LIN {X 0,Y 372.356,Z 524.558,A -85,B 0,C 180,E1 -12798.429,E2 -12798.429} C_VEL
LIN {X 0,Y 373.525,Z 512.398,A -85,B 0,C 180,E1 -12799.938,E2 -12799.938} C_VEL
LIN {X 0,Y 374.797,Z 499.165,A -85,B 0,C 180,E1 -12801.303,E2 -12801.303} C_VEL
LIN {X 0,Y 376.02,Z 484.644,A -85,B 0,C 180,E1 -12802.528,E2 -12802.528} C_VEL
LIN {X 0,Y 377.122,Z 470.65,A -85,B 0,C 180,E1 -12803.473,E2 -12803.473} C_VEL
LIN {X 0,Y 377.997,Z 455.018,A -85,B 0,C 180,E1 -12804.303,E2 -12804.303} C_VEL
LIN {X 0,Y 378.761,Z 440.368,A -85,B 0,C 180,E1 -12804.87,E2 -12804.87} C_VEL
LIN {X 0,Y 379.469,Z 417.557,A -85,B 0,C 180,E1 -12805.468,E2 -12805.468} C_VEL
LIN {X 0,Y 383.226,Z 310.701,A -85,B 0,C 180,E1 -12808.048,E2 -12808.048} C_VEL
LIN {X 0,Y 376.975,Z 295.774,A -85,B 0,C 180,E1 -12808.848,E2 -12808.848} C_VEL
LIN {X 0,Y 369.01,Z 277.788,A -85,B 0,C 180,E1 -12809.879,E2 -12809.879} C_VEL
LIN {X 0,Y 368.929,Z 277.156,A -85,B 0,C 180,E1 -12809.915,E2 -12809.915} C_VEL
LIN {X 0,Y 368.898,Z 277.158,A -85,B 0,C 180,E1 -12813.537,E2 -12813.537} C_VEL
LIN {X 0,Y 368.9,Z 277.154,A -85,B 0,C 180,E1 -12816.854,E2 -12816.854} C_VEL
LIN {X 0,Y 368.906,Z 277.155,A -85,B 0,C 180,E1 -12820.369,E2 -12820.369} C_VEL
LIN {X 0,Y 368.882,Z 277.161,A -85,B 0,C 180,E1 -12823.614,E2 -12823.614} C_VEL
LIN {X 0,Y 368.884,Z 277.157,A -85,B 0,C 180,E1 -12826.694,E2 -12826.694} C_VEL
LIN {X 0,Y 368.909,Z 277.158,A -85,B 0,C 180,E1 -12829.642,E2 -12829.642} C_VEL
LIN {X 0,Y 368.898,Z 277.156,A -85,B 0,C 180,E1 -12833.143,E2 -12833.143} C_VEL
LIN {X 0,Y 368.894,Z 277.156,A -85,B 0,C 180,E1 -12836.46,E2 -12836.46} C_VEL
LIN {X 0,Y 368.909,Z 277.154,A -85,B 0,C 180,E1 -12839.043,E2 -12839.043} C_VEL
LIN {X 0,Y 368.912,Z 277.158,A -85,B 0,C 180,E1 -12841.557,E2 -12841.557} C_VEL
LIN {X 0,Y 368.928,Z 277.153,A -85,B 0,C 180,E1 -12845.221,E2 -12845.221} C_VEL
LIN {X 0,Y 368.915,Z 277.153,A -85,B 0,C 180,E1 -12848.979,E2 -12848.979} C_VEL
LIN {X 0,Y 368.985,Z 277.145,A -85,B 0,C 180,E1 -12852.256,E2 -12852.256} C_VEL
LIN {X 0,Y 369.031,Z 277.139,A -85,B 0,C 180,E1 -12856.226,E2 -12856.226} C_VEL
LIN {X 0,Y 369.061,Z 277.136,A -85,B 0,C 180,E1 -12860.13,E2 -12860.13} C_VEL
LIN {X 0,Y 369.18,Z 277.12,A -85,B 0,C 180,E1 -12862.341,E2 -12862.341} C_VEL
LIN {X 0,Y 369.134,Z 277.125,A -85,B 0,C 180,E1 -12864.536,E2 -12864.536} C_VEL
LIN {X 0,Y 369.308,Z 277.108,A -85,B 0,C 180,E1 -12867.817,E2 -12867.817} C_VEL
LIN {X 0,Y 369.45,Z 277.088,A -85,B 0,C 180,E1 -12869.999,E2 -12869.999} C_VEL
LIN {X 0,Y 369.308,Z 277.105,A -85,B 0,C 180,E1 -12872.18,E2 -12872.18} C_VEL
LIN {X 0,Y 369.197,Z 277.117,A -85,B 0,C 180,E1 -12876.557,E2 -12876.557} C_VEL
LIN {X 0,Y 369.128,Z 277.126,A -85,B 0,C 180,E1 -12878.76,E2 -12878.76} C_VEL
LIN {X 0,Y 368.995,Z 277.144,A -85,B 0,C 180,E1 -12882.092,E2 -12882.092} C_VEL
LIN {X 0,Y 368.987,Z 277.15,A -85,B 0,C 180,E1 -12885.464,E2 -12885.464} C_VEL
LIN {X 0,Y 368.947,Z 277.15,A -85,B 0,C 180,E1 -12888.893,E2 -12888.893} C_VEL
LIN {X 0,Y 368.921,Z 277.155,A -85,B 0,C 180,E1 -12891.149,E2 -12891.149} C_VEL
LIN {X 0,Y 368.237,Z 277.247,A -85,B 0,C 180,E1 -12892.06,E2 -12892.06} C_VEL
LIN {X 0,Y 365.383,Z 277.603,A -85,B 0,C 180,E1 -12893.543,E2 -12893.543} C_VEL
LIN {X 0,Y 362.989,Z 277.896,A -85,B 0,C 180,E1 -12894.741,E2 -12894.741} C_VEL
LIN {X 0,Y 361.982,Z 278.02,A -85,B 0,C 180,E1 -12895.669,E2 -12895.669} C_VEL
LIN {X 0,Y 361.909,Z 278.025,A -85,B 0,C 180,E1 -12895.982,E2 -12895.982} C_VEL
LIN {X 0,Y 361.881,Z 278.032,A -85,B 0,C 180,E1 -12899.084,E2 -12899.084} C_VEL
LIN {X 0,Y 361.835,Z 278.037,A -85,B 0,C 180,E1 -12902.944,E2 -12902.944} C_VEL
LIN {X 0,Y 361.855,Z 278.035,A -85,B 0,C 180,E1 -12905.636,E2 -12905.636} C_VEL
LIN {X 0,Y 361.857,Z 278.035,A -85,B 0,C 180,E1 -12909.026,E2 -12909.026} C_VEL
LIN {X 0,Y 361.823,Z 278.038,A -85,B 0,C 180,E1 -12912.828,E2 -12912.828} C_VEL
LIN {X 0,Y 361.815,Z 278.038,A -85,B 0,C 180,E1 -12915.944,E2 -12915.944} C_VEL
LIN {X 0,Y 361.822,Z 278.043,A -85,B 0,C 180,E1 -12919.244,E2 -12919.244} C_VEL
LIN {X 0,Y 361.849,Z 278.035,A -85,B 0,C 180,E1 -12922.777,E2 -12922.777} C_VEL
LIN {X 0,Y 361.839,Z 278.036,A -85,B 0,C 180,E1 -12925.719,E2 -12925.719} C_VEL
LIN {X 0,Y 361.86,Z 278.033,A -85,B 0,C 180,E1 -12929.672,E2 -12929.672} C_VEL
LIN {X 0,Y 361.939,Z 278.025,A -85,B 0,C 180,E1 -12933.475,E2 -12933.475} C_VEL
LIN {X 0,Y 361.868,Z 278.037,A -85,B 0,C 180,E1 -12937.144,E2 -12937.144} C_VEL
LIN {X 0,Y 361.892,Z 278.03,A -85,B 0,C 180,E1 -12940.724,E2 -12940.724} C_VEL
LIN {X 0,Y 361.919,Z 278.03,A -85,B 0,C 180,E1 -12943.066,E2 -12943.066} C_VEL
LIN {X 0,Y 361.985,Z 278.017,A -85,B 0,C 180,E1 -12946.528,E2 -12946.528} C_VEL
LIN {X 0,Y 362.017,Z 278.012,A -85,B 0,C 180,E1 -12949.939,E2 -12949.939} C_VEL
LIN {X 0,Y 362.147,Z 277.999,A -85,B 0,C 180,E1 -12953.314,E2 -12953.314} C_VEL
LIN {X 0,Y 362.269,Z 277.981,A -85,B 0,C 180,E1 -12957.777,E2 -12957.777} C_VEL
LIN {X 0,Y 362.415,Z 277.962,A -85,B 0,C 180,E1 -12960.001,E2 -12960.001} C_VEL
LIN {X 0,Y 362.267,Z 277.981,A -85,B 0,C 180,E1 -12962.224,E2 -12962.224} C_VEL
LIN {X 0,Y 362.158,Z 277.998,A -85,B 0,C 180,E1 -12966.687,E2 -12966.687} C_VEL
LIN {X 0,Y 362.062,Z 278.013,A -85,B 0,C 180,E1 -12968.934,E2 -12968.934} C_VEL
LIN {X 0,Y 361.948,Z 278.021,A -85,B 0,C 180,E1 -12972.333,E2 -12972.333} C_VEL
LIN {X 0,Y 361.951,Z 278.023,A -85,B 0,C 180,E1 -12974.622,E2 -12974.622} C_VEL
LIN {X 0,Y 361.945,Z 278.021,A -85,B 0,C 180,E1 -12978.101,E2 -12978.101} C_VEL
LIN {X 0,Y 361.851,Z 278.033,A -85,B 0,C 180,E1 -12981.656,E2 -12981.656} C_VEL
LIN {X 0,Y 361.917,Z 278.027,A -85,B 0,C 180,E1 -12985.292,E2 -12985.292} C_VEL
LIN {X 0,Y 361.904,Z 278.026,A -85,B 0,C 180,E1 -12987.78,E2 -12987.78} C_VEL
LIN {X 0,Y 361.837,Z 278.036,A -85,B 0,C 180,E1 -12991.287,E2 -12991.287} C_VEL
LIN {X 0,Y 361.846,Z 278.035,A -85,B 0,C 180,E1 -12994.282,E2 -12994.282} C_VEL
LIN {X 0,Y 361.855,Z 278.034,A -85,B 0,C 180,E1 -12997.224,E2 -12997.224} C_VEL
LIN {X 0,Y 361.828,Z 278.042,A -85,B 0,C 180,E1 -13000.757,E2 -13000.757} C_VEL
LIN {X 0,Y 361.838,Z 278.037,A -85,B 0,C 180,E1 -13004.366,E2 -13004.366} C_VEL
LIN {X 0,Y 361.83,Z 278.035,A -85,B 0,C 180,E1 -13007.57,E2 -13007.57} C_VEL
LIN {X 0,Y 361.864,Z 278.036,A -85,B 0,C 180,E1 -13010.975,E2 -13010.975} C_VEL
LIN {X 0,Y 361.867,Z 278.117,A -85,B 0,C 180,E1 -13012.777,E2 -13012.777} C_VEL
LIN {X 0,Y 365.951,Z 294.107,A -85,B 0,C 180,E1 -13016.158,E2 -13016.158} C_VEL
LIN {X 0,Y 369.838,Z 310.572,A -85,B 0,C 180,E1 -13019.45,E2 -13019.45} C_VEL
LIN {X 0,Y 369.826,Z 313.182,A -85,B 0,C 180,E1 -13019.922,E2 -13019.922} C_VEL
LIN {X 0,Y 376.375,Z 356.911,A -85,B 0,C 180,E1 -13021.56,E2 -13021.56} C_VEL
LIN {X 0,Y 371.811,Z 479.859,A -85,B 0,C 180,E1 -13024.645,E2 -13024.645} C_VEL
LIN {X 0,Y 370.896,Z 495.184,A -85,B 0,C 180,E1 -13025.215,E2 -13025.215} C_VEL
LIN {X 0,Y 369.768,Z 509.984,A -85,B 0,C 180,E1 -13025.971,E2 -13025.971} C_VEL
LIN {X 0,Y 368.493,Z 525.199,A -85,B 0,C 180,E1 -13026.986,E2 -13026.986} C_VEL
LIN {X 0,Y 367.201,Z 538.472,A -85,B 0,C 180,E1 -13028.088,E2 -13028.088} C_VEL
LIN {X 0,Y 365.807,Z 552.139,A -85,B 0,C 180,E1 -13029.476,E2 -13029.476} C_VEL
LIN {X 0,Y 364.498,Z 564.433,A -85,B 0,C 180,E1 -13030.983,E2 -13030.983} C_VEL
LIN {X 0,Y 363.421,Z 575.247,A -85,B 0,C 180,E1 -13032.559,E2 -13032.559} C_VEL
LIN {X 0,Y 362.424,Z 585.017,A -85,B 0,C 180,E1 -13034.249,E2 -13034.249} C_VEL
LIN {X 0,Y 361.728,Z 593.578,A -85,B 0,C 180,E1 -13036.004,E2 -13036.004} C_VEL
LIN {X 0,Y 361.109,Z 601.45,A -85,B 0,C 180,E1 -13037.925,E2 -13037.925} C_VEL
LIN {X 0,Y 360.725,Z 608.122,A -85,B 0,C 180,E1 -13039.903,E2 -13039.903} C_VEL
LIN {X 0,Y 360.555,Z 614.167,A -85,B 0,C 180,E1 -13042.159,E2 -13042.159} C_VEL
LIN {X 0,Y 360.492,Z 618.678,A -85,B 0,C 180,E1 -13044.408,E2 -13044.408} C_VEL
LIN {X 0,Y 360.435,Z 621.759,A -85,B 0,C 180,E1 -13046.648,E2 -13046.648} C_VEL
LIN {X 0,Y 360.564,Z 622.799,A -85,B 0,C 180,E1 -13047.767,E2 -13047.767} C_VEL
LIN {X 0,Y 360.519,Z 623.861,A -85,B 0,C 180,E1 -13050.002,E2 -13050.002} C_VEL
LIN {X 0,Y 360.491,Z 623.607,A -85,B 0,C 180,E1 -13052.236,E2 -13052.236} C_VEL
LIN {X 0,Y 360.403,Z 622.015,A -85,B 0,C 180,E1 -13054.475,E2 -13054.475} C_VEL
LIN {X 0,Y 360.395,Z 619.123,A -85,B 0,C 180,E1 -13056.721,E2 -13056.721} C_VEL
LIN {X 0,Y 360.566,Z 614.896,A -85,B 0,C 180,E1 -13058.972,E2 -13058.972} C_VEL
LIN {X 0,Y 361,Z 609.253,A -85,B 0,C 180,E1 -13061.228,E2 -13061.228} C_VEL
LIN {X 0,Y 361.677,Z 602.075,A -85,B 0,C 180,E1 -13063.486,E2 -13063.486} C_VEL
LIN {X 0,Y 362.806,Z 593.186,A -85,B 0,C 180,E1 -13065.737,E2 -13065.737} C_VEL
LIN {X 0,Y 364.158,Z 583.775,A -85,B 0,C 180,E1 -13067.697,E2 -13067.697} C_VEL
LIN {X 0,Y 365.645,Z 573.556,A -85,B 0,C 180,E1 -13069.491,E2 -13069.491} C_VEL
LIN {X 0,Y 367.627,Z 561.225,A -85,B 0,C 180,E1 -13071.3,E2 -13071.3} C_VEL
LIN {X 0,Y 369.765,Z 547.82,A -85,B 0,C 180,E1 -13072.933,E2 -13072.933} C_VEL
LIN {X 0,Y 372.055,Z 533.098,A -85,B 0,C 180,E1 -13074.408,E2 -13074.408} C_VEL
LIN {X 0,Y 374.237,Z 518.489,A -85,B 0,C 180,E1 -13075.591,E2 -13075.591} C_VEL
LIN {X 0,Y 376.417,Z 502.554,A -85,B 0,C 180,E1 -13076.623,E2 -13076.623} C_VEL
LIN {X 0,Y 378.583,Z 485.245,A -85,B 0,C 180,E1 -13077.466,E2 -13077.466} C_VEL
LIN {X 0,Y 380.092,Z 468.909,A -85,B 0,C 180,E1 -13078.058,E2 -13078.058} C_VEL
LIN {X 0,Y 385.883,Z 394.775,A -85,B 0,C 180,E1 -13080.322,E2 -13080.322} C_VEL
LIN {X 0,Y 389.106,Z 358.696,A -85,B 0,C 180,E1 -13081.484,E2 -13081.484} C_VEL
LIN {X 0,Y 388.296,Z 346.311,A -85,B 0,C 180,E1 -13082.234,E2 -13082.234} C_VEL
LIN {X 0,Y 386.535,Z 330.75,A -85,B 0,C 180,E1 -13083.397,E2 -13083.397} C_VEL
LIN {X 0,Y 383.665,Z 323.796,A -85,B 0,C 180,E1 -13084.421,E2 -13084.421} C_VEL
LIN {X 0,Y 381.231,Z 318.55,A -85,B 0,C 180,E1 -13085.337,E2 -13085.337} C_VEL
LIN {X 0,Y 378.301,Z 312.803,A -85,B 0,C 180,E1 -13086.548,E2 -13086.548} C_VEL
LIN {X 0,Y 374.397,Z 305.694,A -85,B 0,C 180,E1 -13088.473,E2 -13088.473} C_VEL
LIN {X 0,Y 370.905,Z 299.971,A -85,B 0,C 180,E1 -13090.782,E2 -13090.782} C_VEL
LIN {X 0,Y 369.189,Z 296.566,A -85,B 0,C 180,E1 -13092.669,E2 -13092.669} C_VEL
LIN {X 0,Y 368.787,Z 295.464,A -85,B 0,C 180,E1 -13093.6,E2 -13093.6} C_VEL
LIN {X 0,Y 368.258,Z 294.192,A -85,B 0,C 180,E1 -13095.439,E2 -13095.439} C_VEL
LIN {X 0,Y 368.708,Z 294.364,A -85,B 0,C 180,E1 -13097.364,E2 -13097.364} C_VEL
LIN {X 0,Y 370.91,Z 296.011,A -85,B 0,C 180,E1 -13099.891,E2 -13099.891} C_VEL
LIN {X 0,Y 372.199,Z 297.038,A -85,B 0,C 180,E1 -13100.825,E2 -13100.825} C_VEL
LIN {X 0,Y 375.738,Z 300.987,A -85,B 0,C 180,E1 -13102.863,E2 -13102.863} C_VEL
LIN {X 0,Y 379.159,Z 305.289,A -85,B 0,C 180,E1 -13104.391,E2 -13104.391} C_VEL
LIN {X 0,Y 382.506,Z 310.037,A -85,B 0,C 180,E1 -13105.673,E2 -13105.673} C_VEL
LIN {X 0,Y 386.077,Z 315.376,A -85,B 0,C 180,E1 -13106.865,E2 -13106.865} C_VEL
LIN {X 0,Y 390.641,Z 323.626,A -85,B 0,C 180,E1 -13108.26,E2 -13108.26} C_VEL
LIN {X 0,Y 391.487,Z 325.432,A -85,B 0,C 180,E1 -13108.513,E2 -13108.513} C_VEL
LIN {X 0,Y 383.852,Z 405.157,A -85,B 0,C 180,E1 -13111.049,E2 -13111.049} C_VEL
LIN {X 0,Y 380.62,Z 447.423,A -85,B 0,C 180,E1 -13112.387,E2 -13112.387} C_VEL
LIN {X 0,Y 379.204,Z 462.75,A -85,B 0,C 180,E1 -13113.077,E2 -13113.077} C_VEL
LIN {X 0,Y 377.435,Z 478.879,A -85,B 0,C 180,E1 -13114.05,E2 -13114.05} C_VEL
LIN {X 0,Y 375.724,Z 492.725,A -85,B 0,C 180,E1 -13115.11,E2 -13115.11} C_VEL
LIN {X 0,Y 373.879,Z 505.632,A -85,B 0,C 180,E1 -13116.309,E2 -13116.309} C_VEL
LIN {X 0,Y 371.825,Z 518.795,A -85,B 0,C 180,E1 -13117.788,E2 -13117.788} C_VEL
LIN {X 0,Y 370.029,Z 528.933,A -85,B 0,C 180,E1 -13119.137,E2 -13119.137} C_VEL
LIN {X 0,Y 368.265,Z 539.317,A -85,B 0,C 180,E1 -13120.779,E2 -13120.779} C_VEL
LIN {X 0,Y 366.473,Z 549.487,A -85,B 0,C 180,E1 -13122.707,E2 -13122.707} C_VEL
LIN {X 0,Y 364.854,Z 557.896,A -85,B 0,C 180,E1 -13124.624,E2 -13124.624} C_VEL
LIN {X 0,Y 363.668,Z 564.97,A -85,B 0,C 180,E1 -13126.59,E2 -13126.59} C_VEL
LIN {X 0,Y 362.517,Z 571.438,A -85,B 0,C 180,E1 -13128.821,E2 -13128.821} C_VEL
LIN {X 0,Y 361.765,Z 576.407,A -85,B 0,C 180,E1 -13131.058,E2 -13131.058} C_VEL
LIN {X 0,Y 361.195,Z 580.029,A -85,B 0,C 180,E1 -13133.295,E2 -13133.295} C_VEL
LIN {X 0,Y 360.877,Z 582.365,A -85,B 0,C 180,E1 -13135.531,E2 -13135.531} C_VEL
LIN {X 0,Y 360.694,Z 583.454,A -85,B 0,C 180,E1 -13137.766,E2 -13137.766} C_VEL
LIN {X 0,Y 360.524,Z 583.282,A -85,B 0,C 180,E1 -13139.999,E2 -13139.999} C_VEL
LIN {X 0,Y 360.61,Z 581.862,A -85,B 0,C 180,E1 -13142.233,E2 -13142.233} C_VEL
LIN {X 0,Y 360.609,Z 579.19,A -85,B 0,C 180,E1 -13144.47,E2 -13144.47} C_VEL
LIN {X 0,Y 360.827,Z 574.99,A -85,B 0,C 180,E1 -13146.806,E2 -13146.806} C_VEL
LIN {X 0,Y 361.116,Z 569.776,A -85,B 0,C 180,E1 -13148.956,E2 -13148.956} C_VEL
LIN {X 0,Y 361.608,Z 562.801,A -85,B 0,C 180,E1 -13151.206,E2 -13151.206} C_VEL
LIN {X 0,Y 362.378,Z 555.243,A -85,B 0,C 180,E1 -13153.171,E2 -13153.171} C_VEL
LIN {X 0,Y 363.207,Z 546.104,A -85,B 0,C 180,E1 -13155.142,E2 -13155.142} C_VEL
LIN {X 0,Y 364.364,Z 535.081,A -85,B 0,C 180,E1 -13157.105,E2 -13157.105} C_VEL
LIN {X 0,Y 365.534,Z 523.732,A -85,B 0,C 180,E1 -13158.786,E2 -13158.786} C_VEL
LIN {X 0,Y 366.761,Z 511.326,A -85,B 0,C 180,E1 -13160.322,E2 -13160.322} C_VEL
LIN {X 0,Y 368.079,Z 497.791,A -85,B 0,C 180,E1 -13161.711,E2 -13161.711} C_VEL
LIN {X 0,Y 369.19,Z 484.653,A -85,B 0,C 180,E1 -13162.82,E2 -13162.82} C_VEL
LIN {X 0,Y 370.313,Z 470.577,A -85,B 0,C 180,E1 -13163.783,E2 -13163.783} C_VEL
LIN {X 0,Y 371.208,Z 455.124,A -85,B 0,C 180,E1 -13164.614,E2 -13164.614} C_VEL
LIN {X 0,Y 372.028,Z 439.672,A -85,B 0,C 180,E1 -13165.216,E2 -13165.216} C_VEL
LIN {X 0,Y 372.982,Z 410.158,A -85,B 0,C 180,E1 -13165.981,E2 -13165.981} C_VEL
LIN {X 0,Y 376.663,Z 312.659,A -85,B 0,C 180,E1 -13168.402,E2 -13168.402} C_VEL
LIN {X 0,Y 371.332,Z 299.862,A -85,B 0,C 180,E1 -13169.098,E2 -13169.098} C_VEL
LIN {X 0,Y 361.953,Z 278.543,A -85,B 0,C 180,E1 -13170.344,E2 -13170.344} C_VEL
LIN {X 0,Y 361.888,Z 278.033,A -85,B 0,C 180,E1 -13170.402,E2 -13170.402} C_VEL
LIN {X 0,Y 361.855,Z 278.035,A -85,B 0,C 180,E1 -13174.279,E2 -13174.279} C_VEL
LIN {X 0,Y 361.861,Z 278.032,A -85,B 0,C 180,E1 -13177.221,E2 -13177.221} C_VEL
LIN {X 0,Y 361.829,Z 278.035,A -85,B 0,C 180,E1 -13180.753,E2 -13180.753} C_VEL
LIN {X 0,Y 361.816,Z 278.038,A -85,B 0,C 180,E1 -13184.367,E2 -13184.367} C_VEL
LIN {X 0,Y 361.835,Z 278.038,A -85,B 0,C 180,E1 -13187.566,E2 -13187.566} C_VEL
LIN {X 0,Y 361.866,Z 278.031,A -85,B 0,C 180,E1 -13190.972,E2 -13190.972} C_VEL
LIN {X 0,Y 361.871,Z 278.03,A -85,B 0,C 180,E1 -13194.654,E2 -13194.654} C_VEL
LIN {X 0,Y 361.834,Z 278.036,A -85,B 0,C 180,E1 -13198.369,E2 -13198.369} C_VEL
LIN {X 0,Y 361.862,Z 278.032,A -85,B 0,C 180,E1 -13200.95,E2 -13200.95} C_VEL
LIN {X 0,Y 361.886,Z 278.028,A -85,B 0,C 180,E1 -13204.705,E2 -13204.705} C_VEL
LIN {X 0,Y 361.856,Z 278.033,A -85,B 0,C 180,E1 -13208.343,E2 -13208.343} C_VEL
LIN {X 0,Y 361.915,Z 278.027,A -85,B 0,C 180,E1 -13212.083,E2 -13212.083} C_VEL
LIN {X 0,Y 361.956,Z 278.023,A -85,B 0,C 180,E1 -13215.378,E2 -13215.378} C_VEL
LIN {X 0,Y 361.965,Z 278.019,A -85,B 0,C 180,E1 -13218.803,E2 -13218.803} C_VEL
LIN {X 0,Y 362.143,Z 277.997,A -85,B 0,C 180,E1 -13222.191,E2 -13222.191} C_VEL
LIN {X 0,Y 362.108,Z 278.001,A -85,B 0,C 180,E1 -13224.43,E2 -13224.43} C_VEL
LIN {X 0,Y 362.272,Z 277.984,A -85,B 0,C 180,E1 -13227.775,E2 -13227.775} C_VEL
LIN {X 0,Y 362.419,Z 277.964,A -85,B 0,C 180,E1 -13229.998,E2 -13229.998} C_VEL
LIN {X 0,Y 362.272,Z 277.981,A -85,B 0,C 180,E1 -13232.222,E2 -13232.222} C_VEL
LIN {X 0,Y 362.161,Z 277.994,A -85,B 0,C 180,E1 -13236.685,E2 -13236.685} C_VEL
LIN {X 0,Y 362.064,Z 278.007,A -85,B 0,C 180,E1 -13238.932,E2 -13238.932} C_VEL
LIN {X 0,Y 361.95,Z 278.02,A -85,B 0,C 180,E1 -13242.331,E2 -13242.331} C_VEL
LIN {X 0,Y 361.951,Z 278.02,A -85,B 0,C 180,E1 -13244.619,E2 -13244.619} C_VEL
LIN {X 0,Y 361.945,Z 278.022,A -85,B 0,C 180,E1 -13248.098,E2 -13248.098} C_VEL
LIN {X 0,Y 361.882,Z 278.033,A -85,B 0,C 180,E1 -13251.652,E2 -13251.652} C_VEL
LIN {X 0,Y 361.916,Z 278.03,A -85,B 0,C 180,E1 -13255.289,E2 -13255.289} C_VEL
LIN {X 0,Y 361.909,Z 278.025,A -85,B 0,C 180,E1 -13255.982,E2 -13255.982} C_VEL
LIN {X 0,Y 361.251,Z 278.111,A -85,B 0,C 180,E1 -13256.911,E2 -13256.911} C_VEL
LIN {X 0,Y 358.342,Z 278.47,A -85,B 0,C 180,E1 -13258.42,E2 -13258.42} C_VEL
LIN {X 0,Y 355.883,Z 278.78,A -85,B 0,C 180,E1 -13259.642,E2 -13259.642} C_VEL
LIN {X 0,Y 354.851,Z 278.905,A -85,B 0,C 180,E1 -13260.588,E2 -13260.588} C_VEL
LIN {X 0,Y 354.782,Z 278.915,A -85,B 0,C 180,E1 -13260.908,E2 -13260.908} C_VEL
LIN {X 0,Y 354.793,Z 278.915,A -85,B 0,C 180,E1 -13263.701,E2 -13263.701} C_VEL
LIN {X 0,Y 354.787,Z 278.913,A -85,B 0,C 180,E1 -13266.458,E2 -13266.458} C_VEL
LIN {X 0,Y 354.81,Z 278.915,A -85,B 0,C 180,E1 -13269.423,E2 -13269.423} C_VEL
LIN {X 0,Y 354.775,Z 278.916,A -85,B 0,C 180,E1 -13272.867,E2 -13272.867} C_VEL
LIN {X 0,Y 354.762,Z 278.916,A -85,B 0,C 180,E1 -13276.105,E2 -13276.105} C_VEL
LIN {X 0,Y 354.774,Z 278.92,A -85,B 0,C 180,E1 -13279.179,E2 -13279.179} C_VEL
LIN {X 0,Y 354.793,Z 278.912,A -85,B 0,C 180,E1 -13282.402,E2 -13282.402} C_VEL
LIN {X 0,Y 354.797,Z 278.915,A -85,B 0,C 180,E1 -13284.941,E2 -13284.941} C_VEL
LIN {X 0,Y 354.778,Z 278.914,A -85,B 0,C 180,E1 -13288.405,E2 -13288.405} C_VEL
LIN {X 0,Y 354.835,Z 278.909,A -85,B 0,C 180,E1 -13291.619,E2 -13291.619} C_VEL
LIN {X 0,Y 354.884,Z 278.9,A -85,B 0,C 180,E1 -13294.173,E2 -13294.173} C_VEL
LIN {X 0,Y 354.802,Z 278.911,A -85,B 0,C 180,E1 -13297.893,E2 -13297.893} C_VEL
LIN {X 0,Y 354.908,Z 278.898,A -85,B 0,C 180,E1 -13301.892,E2 -13301.892} C_VEL
LIN {X 0,Y 354.929,Z 278.895,A -85,B 0,C 180,E1 -13305.982,E2 -13305.982} C_VEL
LIN {X 0,Y 354.964,Z 278.891,A -85,B 0,C 180,E1 -13309.737,E2 -13309.737} C_VEL
LIN {X 0,Y 355.111,Z 278.877,A -85,B 0,C 180,E1 -13313.181,E2 -13313.181} C_VEL
LIN {X 0,Y 355.232,Z 278.858,A -85,B 0,C 180,E1 -13317.733,E2 -13317.733} C_VEL
LIN {X 0,Y 355.385,Z 278.838,A -85,B 0,C 180,E1 -13320.001,E2 -13320.001} C_VEL
LIN {X 0,Y 355.23,Z 278.858,A -85,B 0,C 180,E1 -13322.269,E2 -13322.269} C_VEL
LIN {X 0,Y 355.124,Z 278.875,A -85,B 0,C 180,E1 -13326.82,E2 -13326.82} C_VEL
LIN {X 0,Y 355.004,Z 278.89,A -85,B 0,C 180,E1 -13329.113,E2 -13329.113} C_VEL
LIN {X 0,Y 354.91,Z 278.9,A -85,B 0,C 180,E1 -13332.582,E2 -13332.582} C_VEL
LIN {X 0,Y 354.878,Z 278.901,A -85,B 0,C 180,E1 -13336.097,E2 -13336.097} C_VEL
LIN {X 0,Y 354.891,Z 278.902,A -85,B 0,C 180,E1 -13338.473,E2 -13338.473} C_VEL
LIN {X 0,Y 354.807,Z 278.91,A -85,B 0,C 180,E1 -13342.109,E2 -13342.109} C_VEL
LIN {X 0,Y 354.889,Z 278.9,A -85,B 0,C 180,E1 -13345.829,E2 -13345.829} C_VEL
LIN {X 0,Y 354.845,Z 278.906,A -85,B 0,C 180,E1 -13349.68,E2 -13349.68} C_VEL
LIN {X 0,Y 354.798,Z 278.911,A -85,B 0,C 180,E1 -13353.704,E2 -13353.704} C_VEL
LIN {X 0,Y 354.789,Z 278.915,A -85,B 0,C 180,E1 -13356.461,E2 -13356.461} C_VEL
LIN {X 0,Y 354.817,Z 278.91,A -85,B 0,C 180,E1 -13359.425,E2 -13359.425} C_VEL
LIN {X 0,Y 354.781,Z 278.919,A -85,B 0,C 180,E1 -13362.869,E2 -13362.869} C_VEL
LIN {X 0,Y 354.762,Z 278.917,A -85,B 0,C 180,E1 -13366.106,E2 -13366.106} C_VEL
LIN {X 0,Y 354.782,Z 278.918,A -85,B 0,C 180,E1 -13369.181,E2 -13369.181} C_VEL
LIN {X 0,Y 354.847,Z 278.966,A -85,B 0,C 180,E1 -13372.361,E2 -13372.361} C_VEL
LIN {X 0,Y 359.247,Z 296.405,A -85,B 0,C 180,E1 -13376.116,E2 -13376.116} C_VEL
LIN {X 0,Y 362.932,Z 311.997,A -85,B 0,C 180,E1 -13379.288,E2 -13379.288} C_VEL
LIN {X 0,Y 363.077,Z 313.226,A -85,B 0,C 180,E1 -13379.472,E2 -13379.472} C_VEL
LIN {X 0,Y 369.741,Z 357.719,A -85,B 0,C 180,E1 -13381.181,E2 -13381.181} C_VEL
LIN {X 0,Y 365.017,Z 479.813,A -85,B 0,C 180,E1 -13384.33,E2 -13384.33} C_VEL
LIN {X 0,Y 363.984,Z 496.194,A -85,B 0,C 180,E1 -13384.968,E2 -13384.968} C_VEL
LIN {X 0,Y 362.839,Z 511.005,A -85,B 0,C 180,E1 -13385.761,E2 -13385.761} C_VEL
LIN {X 0,Y 361.493,Z 526.191,A -85,B 0,C 180,E1 -13386.818,E2 -13386.818} C_VEL
LIN {X 0,Y 360.19,Z 539.216,A -85,B 0,C 180,E1 -13387.94,E2 -13387.94} C_VEL
LIN {X 0,Y 358.772,Z 552.689,A -85,B 0,C 180,E1 -13389.355,E2 -13389.355} C_VEL
LIN {X 0,Y 357.382,Z 565.219,A -85,B 0,C 180,E1 -13390.945,E2 -13390.945} C_VEL
LIN {X 0,Y 356.327,Z 575.531,A -85,B 0,C 180,E1 -13392.497,E2 -13392.497} C_VEL
LIN {X 0,Y 355.332,Z 585.239,A -85,B 0,C 180,E1 -13394.221,E2 -13394.221} C_VEL
LIN {X 0,Y 354.5,Z 594.861,A -85,B 0,C 180,E1 -13396.273,E2 -13396.273} C_VEL
LIN {X 0,Y 353.985,Z 602.563,A -85,B 0,C 180,E1 -13398.26,E2 -13398.26} C_VEL
LIN {X 0,Y 353.594,Z 608.931,A -85,B 0,C 180,E1 -13400.275,E2 -13400.275} C_VEL
LIN {X 0,Y 353.48,Z 613.391,A -85,B 0,C 180,E1 -13402.001,E2 -13402.001} C_VEL
LIN {X 0,Y 353.43,Z 618.004,A -85,B 0,C 180,E1 -13404.296,E2 -13404.296} C_VEL
LIN {X 0,Y 353.348,Z 621.175,A -85,B 0,C 180,E1 -13406.581,E2 -13406.581} C_VEL
LIN {X 0,Y 353.482,Z 622.259,A -85,B 0,C 180,E1 -13407.723,E2 -13407.723} C_VEL
LIN {X 0,Y 353.454,Z 623.4,A -85,B 0,C 180,E1 -13410.002,E2 -13410.002} C_VEL
LIN {X 0,Y 353.467,Z 623.464,A -85,B 0,C 180,E1 -13411.141,E2 -13411.141} C_VEL
LIN {X 0,Y 353.305,Z 622.586,A -85,B 0,C 180,E1 -13413.423,E2 -13413.423} C_VEL
LIN {X 0,Y 353.312,Z 620.419,A -85,B 0,C 180,E1 -13415.71,E2 -13415.71} C_VEL
LIN {X 0,Y 353.396,Z 616.945,A -85,B 0,C 180,E1 -13418.004,E2 -13418.004} C_VEL
LIN {X 0,Y 353.647,Z 612.107,A -85,B 0,C 180,E1 -13420.305,E2 -13420.305} C_VEL
LIN {X 0,Y 354.276,Z 605.801,A -85,B 0,C 180,E1 -13422.606,E2 -13422.606} C_VEL
LIN {X 0,Y 355.257,Z 597.902,A -85,B 0,C 180,E1 -13424.904,E2 -13424.904} C_VEL
LIN {X 0,Y 356.476,Z 589.531,A -85,B 0,C 180,E1 -13426.907,E2 -13426.907} C_VEL
LIN {X 0,Y 358.053,Z 579.559,A -85,B 0,C 180,E1 -13428.898,E2 -13428.898} C_VEL
LIN {X 0,Y 360.045,Z 567.668,A -85,B 0,C 180,E1 -13430.871,E2 -13430.871} C_VEL
LIN {X 0,Y 362.343,Z 554.497,A -85,B 0,C 180,E1 -13432.676,E2 -13432.676} C_VEL
LIN {X 0,Y 364.583,Z 541.247,A -85,B 0,C 180,E1 -13434.183,E2 -13434.183} C_VEL
LIN {X 0,Y 366.859,Z 527.358,A -85,B 0,C 180,E1 -13435.493,E2 -13435.493} C_VEL
LIN {X 0,Y 369.401,Z 511.331,A -85,B 0,C 180,E1 -13436.711,E2 -13436.711} C_VEL
LIN {X 0,Y 371.72,Z 495.021,A -85,B 0,C 180,E1 -13437.672,E2 -13437.672} C_VEL
LIN {X 0,Y 373.743,Z 478.107,A -85,B 0,C 180,E1 -13438.425,E2 -13438.425} C_VEL
LIN {X 0,Y 376.103,Z 449.941,A -85,B 0,C 180,E1 -13439.338,E2 -13439.338} C_VEL
LIN {X 0,Y 382.639,Z 377.508,A -85,B 0,C 180,E1 -13441.652,E2 -13441.652} C_VEL
LIN {X 0,Y 384.308,Z 359.927,A -85,B 0,C 180,E1 -13442.25,E2 -13442.25} C_VEL
LIN {X 0,Y 383.617,Z 347.484,A -85,B 0,C 180,E1 -13443.046,E2 -13443.046} C_VEL
LIN {X 0,Y 382.35,Z 334.467,A -85,B 0,C 180,E1 -13444.056,E2 -13444.056} C_VEL
LIN {X 0,Y 379.643,Z 327.893,A -85,B 0,C 180,E1 -13445.103,E2 -13445.103} C_VEL
LIN {X 0,Y 377.831,Z 323.802,A -85,B 0,C 180,E1 -13445.855,E2 -13445.855} C_VEL
LIN {X 0,Y 375.368,Z 318.639,A -85,B 0,C 180,E1 -13446.97,E2 -13446.97} C_VEL
LIN {X 0,Y 371.788,Z 311.774,A -85,B 0,C 180,E1 -13448.882,E2 -13448.882} C_VEL
LIN {X 0,Y 368.72,Z 306.358,A -85,B 0,C 180,E1 -13451.127,E2 -13451.127} C_VEL
LIN {X 0,Y 367.199,Z 303.09,A -85,B 0,C 180,E1 -13453.028,E2 -13453.028} C_VEL
LIN {X 0,Y 366.551,Z 301.266,A -85,B 0,C 180,E1 -13454.994,E2 -13454.994} C_VEL
LIN {X 0,Y 366.72,Z 301.084,A -85,B 0,C 180,E1 -13456.741,E2 -13456.741} C_VEL
LIN {X 0,Y 368.262,Z 302.294,A -85,B 0,C 180,E1 -13459.111,E2 -13459.111} C_VEL
LIN {X 0,Y 370.12,Z 303.682,A -85,B 0,C 180,E1 -13460.616,E2 -13460.616} C_VEL
LIN {X 0,Y 373.318,Z 307.382,A -85,B 0,C 180,E1 -13462.566,E2 -13462.566} C_VEL
LIN {X 0,Y 376.504,Z 311.606,A -85,B 0,C 180,E1 -13464.091,E2 -13464.091} C_VEL
LIN {X 0,Y 379.61,Z 316.139,A -85,B 0,C 180,E1 -13465.348,E2 -13465.348} C_VEL
LIN {X 0,Y 383.164,Z 321.892,A -85,B 0,C 180,E1 -13466.614,E2 -13466.614} C_VEL
LIN {X 0,Y 386.765,Z 328.599,A -85,B 0,C 180,E1 -13467.781,E2 -13467.781} C_VEL
LIN {X 0,Y 378.774,Z 405.947,A -85,B 0,C 180,E1 -13470.318,E2 -13470.318} C_VEL
LIN {X 0,Y 375.238,Z 447.944,A -85,B 0,C 180,E1 -13471.693,E2 -13471.693} C_VEL
LIN {X 0,Y 373.676,Z 463.454,A -85,B 0,C 180,E1 -13472.41,E2 -13472.41} C_VEL
LIN {X 0,Y 371.911,Z 478.54,A -85,B 0,C 180,E1 -13473.332,E2 -13473.332} C_VEL
LIN {X 0,Y 370.058,Z 492.413,A -85,B 0,C 180,E1 -13474.401,E2 -13474.401} C_VEL
LIN {X 0,Y 367.87,Z 506.681,A -85,B 0,C 180,E1 -13475.747,E2 -13475.747} C_VEL
LIN {X 0,Y 365.818,Z 518.802,A -85,B 0,C 180,E1 -13477.135,E2 -13477.135} C_VEL
LIN {X 0,Y 363.934,Z 528.802,A -85,B 0,C 180,E1 -13478.474,E2 -13478.474} C_VEL
LIN {X 0,Y 361.986,Z 539.255,A -85,B 0,C 180,E1 -13480.137,E2 -13480.137} C_VEL
LIN {X 0,Y 360.089,Z 549.475,A -85,B 0,C 180,E1 -13482.097,E2 -13482.097} C_VEL
LIN {X 0,Y 358.33,Z 558.016,A -85,B 0,C 180,E1 -13484.062,E2 -13484.062} C_VEL
LIN {X 0,Y 357.116,Z 564.203,A -85,B 0,C 180,E1 -13485.758,E2 -13485.758} C_VEL
LIN {X 0,Y 355.825,Z 570.935,A -85,B 0,C 180,E1 -13488.03,E2 -13488.03} C_VEL
LIN {X 0,Y 355.027,Z 576.129,A -85,B 0,C 180,E1 -13490.312,E2 -13490.312} C_VEL
LIN {X 0,Y 354.262,Z 580.158,A -85,B 0,C 180,E1 -13492.72,E2 -13492.72} C_VEL
LIN {X 0,Y 353.85,Z 581.984,A -85,B 0,C 180,E1 -13494.3,E2 -13494.3} C_VEL
LIN {X 0,Y 353.789,Z 583.588,A -85,B 0,C 180,E1 -13496.583,E2 -13496.583} C_VEL
LIN {X 0,Y 353.51,Z 583.979,A -85,B 0,C 180,E1 -13498.86,E2 -13498.86} C_VEL
LIN {X 0,Y 353.488,Z 583.09,A -85,B 0,C 180,E1 -13501.138,E2 -13501.138} C_VEL
LIN {X 0,Y 353.493,Z 580.947,A -85,B 0,C 180,E1 -13503.418,E2 -13503.418} C_VEL
LIN {X 0,Y 353.645,Z 577.51,A -85,B 0,C 180,E1 -13505.702,E2 -13505.702} C_VEL
LIN {X 0,Y 353.887,Z 572.701,A -85,B 0,C 180,E1 -13507.99,E2 -13507.99} C_VEL
LIN {X 0,Y 354.301,Z 566.395,A -85,B 0,C 180,E1 -13510.283,E2 -13510.283} C_VEL
LIN {X 0,Y 354.975,Z 559.497,A -85,B 0,C 180,E1 -13512.287,E2 -13512.287} C_VEL
LIN {X 0,Y 355.702,Z 551.855,A -85,B 0,C 180,E1 -13514.137,E2 -13514.137} C_VEL
LIN {X 0,Y 356.579,Z 542.611,A -85,B 0,C 180,E1 -13516.017,E2 -13516.017} C_VEL
LIN {X 0,Y 357.628,Z 532.582,A -85,B 0,C 180,E1 -13517.733,E2 -13517.733} C_VEL
LIN {X 0,Y 358.937,Z 520.654,A -85,B 0,C 180,E1 -13519.441,E2 -13519.441} C_VEL
LIN {X 0,Y 360.104,Z 508.85,A -85,B 0,C 180,E1 -13520.864,E2 -13520.864} C_VEL
LIN {X 0,Y 361.306,Z 496.246,A -85,B 0,C 180,E1 -13522.139,E2 -13522.139} C_VEL
LIN {X 0,Y 362.526,Z 482.752,A -85,B 0,C 180,E1 -13523.264,E2 -13523.264} C_VEL
LIN {X 0,Y 363.67,Z 467.52,A -85,B 0,C 180,E1 -13524.28,E2 -13524.28} C_VEL
LIN {X 0,Y 364.616,Z 451.666,A -85,B 0,C 180,E1 -13525.089,E2 -13525.089} C_VEL
LIN {X 0,Y 365.374,Z 436.556,A -85,B 0,C 180,E1 -13525.643,E2 -13525.643} C_VEL
LIN {X 0,Y 370.074,Z 314.289,A -85,B 0,C 180,E1 -13528.773,E2 -13528.773} C_VEL
LIN {X 0,Y 362.59,Z 296.978,A -85,B 0,C 180,E1 -13529.76,E2 -13529.76} C_VEL
LIN {X 0,Y 354.945,Z 279.487,A -85,B 0,C 180,E1 -13530.812,E2 -13530.812} C_VEL
LIN {X 0,Y 354.836,Z 278.91,A -85,B 0,C 180,E1 -13530.889,E2 -13530.889} C_VEL
LIN {X 0,Y 354.808,Z 278.914,A -85,B 0,C 180,E1 -13533.7,E2 -13533.7} C_VEL
LIN {X 0,Y 354.796,Z 278.913,A -85,B 0,C 180,E1 -13536.458,E2 -13536.458} C_VEL
LIN {X 0,Y 354.799,Z 278.913,A -85,B 0,C 180,E1 -13539.417,E2 -13539.417} C_VEL
LIN {X 0,Y 354.785,Z 278.913,A -85,B 0,C 180,E1 -13542.865,E2 -13542.865} C_VEL
LIN {X 0,Y 354.766,Z 278.919,A -85,B 0,C 180,E1 -13546.102,E2 -13546.102} C_VEL
LIN {X 0,Y 354.786,Z 278.914,A -85,B 0,C 180,E1 -13549.177,E2 -13549.177} C_VEL
LIN {X 0,Y 354.804,Z 278.911,A -85,B 0,C 180,E1 -13552.401,E2 -13552.401} C_VEL
LIN {X 0,Y 354.809,Z 278.91,A -85,B 0,C 180,E1 -13554.939,E2 -13554.939} C_VEL
LIN {X 0,Y 354.79,Z 278.913,A -85,B 0,C 180,E1 -13558.404,E2 -13558.404} C_VEL
LIN {X 0,Y 354.798,Z 278.916,A -85,B 0,C 180,E1 -13561.613,E2 -13561.613} C_VEL
LIN {X 0,Y 354.846,Z 278.909,A -85,B 0,C 180,E1 -13565.421,E2 -13565.421} C_VEL
LIN {X 0,Y 354.822,Z 278.909,A -85,B 0,C 180,E1 -13569.111,E2 -13569.111} C_VEL
LIN {X 0,Y 354.875,Z 278.902,A -85,B 0,C 180,E1 -13572.717,E2 -13572.717} C_VEL
LIN {X 0,Y 354.945,Z 278.894,A -85,B 0,C 180,E1 -13576.253,E2 -13576.253} C_VEL
LIN {X 0,Y 354.971,Z 278.895,A -85,B 0,C 180,E1 -13579.734,E2 -13579.734} C_VEL
LIN {X 0,Y 355.107,Z 278.875,A -85,B 0,C 180,E1 -13582.035,E2 -13582.035} C_VEL
LIN {X 0,Y 355.083,Z 278.876,A -85,B 0,C 180,E1 -13584.319,E2 -13584.319} C_VEL
LIN {X 0,Y 355.235,Z 278.861,A -85,B 0,C 180,E1 -13587.731,E2 -13587.731} C_VEL
LIN {X 0,Y 355.389,Z 278.84,A -85,B 0,C 180,E1 -13589.998,E2 -13589.998} C_VEL
LIN {X 0,Y 355.235,Z 278.857,A -85,B 0,C 180,E1 -13592.266,E2 -13592.266} C_VEL
LIN {X 0,Y 355.127,Z 278.871,A -85,B 0,C 180,E1 -13596.818,E2 -13596.818} C_VEL
LIN {X 0,Y 355.006,Z 278.888,A -85,B 0,C 180,E1 -13599.111,E2 -13599.111} C_VEL
LIN {X 0,Y 354.911,Z 278.897,A -85,B 0,C 180,E1 -13602.58,E2 -13602.58} C_VEL
LIN {X 0,Y 354.878,Z 278.902,A -85,B 0,C 180,E1 -13606.095,E2 -13606.095} C_VEL
LIN {X 0,Y 354.89,Z 278.9,A -85,B 0,C 180,E1 -13608.471,E2 -13608.471} C_VEL
LIN {X 0,Y 354.824,Z 278.909,A -85,B 0,C 180,E1 -13612.105,E2 -13612.105} C_VEL
LIN {X 0,Y 354.877,Z 278.903,A -85,B 0,C 180,E1 -13615.972,E2 -13615.972} C_VEL
LIN {X 0,Y 354.805,Z 278.914,A -85,B 0,C 180,E1 -13619.681,E2 -13619.681} C_VEL
LIN {X 0,Y 354.782,Z 278.915,A -85,B 0,C 180,E1 -13620.908,E2 -13620.908} C_VEL
LIN {X 0,Y 354.168,Z 278.997,A -85,B 0,C 180,E1 -13621.856,E2 -13621.856} C_VEL
LIN {X 0,Y 351.378,Z 279.348,A -85,B 0,C 180,E1 -13623.398,E2 -13623.398} C_VEL
LIN {X 0,Y 348.961,Z 279.646,A -85,B 0,C 180,E1 -13624.646,E2 -13624.646} C_VEL
LIN {X 0,Y 347.88,Z 279.777,A -85,B 0,C 180,E1 -13625.611,E2 -13625.611} C_VEL
LIN {X 0,Y 347.77,Z 279.788,A -85,B 0,C 180,E1 -13625.938,E2 -13625.938} C_VEL
LIN {X 0,Y 347.74,Z 279.792,A -85,B 0,C 180,E1 -13628.792,E2 -13628.792} C_VEL
LIN {X 0,Y 347.737,Z 279.792,A -85,B 0,C 180,E1 -13631.83,E2 -13631.83} C_VEL
LIN {X 0,Y 347.753,Z 279.792,A -85,B 0,C 180,E1 -13635.016,E2 -13635.016} C_VEL
LIN {X 0,Y 347.736,Z 279.791,A -85,B 0,C 180,E1 -13638.397,E2 -13638.397} C_VEL
LIN {X 0,Y 347.759,Z 279.788,A -85,B 0,C 180,E1 -13642.011,E2 -13642.011} C_VEL
LIN {X 0,Y 347.73,Z 279.795,A -85,B 0,C 180,E1 -13645.536,E2 -13645.536} C_VEL
LIN {X 0,Y 347.749,Z 279.791,A -85,B 0,C 180,E1 -13649.654,E2 -13649.654} C_VEL
LIN {X 0,Y 347.836,Z 279.781,A -85,B 0,C 180,E1 -13652.745,E2 -13652.745} C_VEL
LIN {X 0,Y 347.771,Z 279.787,A -85,B 0,C 180,E1 -13656.162,E2 -13656.162} C_VEL
LIN {X 0,Y 347.792,Z 279.784,A -85,B 0,C 180,E1 -13659.909,E2 -13659.909} C_VEL
LIN {X 0,Y 347.852,Z 279.777,A -85,B 0,C 180,E1 -13662.36,E2 -13662.36} C_VEL
LIN {X 0,Y 347.884,Z 279.773,A -85,B 0,C 180,E1 -13665.971,E2 -13665.971} C_VEL
LIN {X 0,Y 347.915,Z 279.771,A -85,B 0,C 180,E1 -13669.526,E2 -13669.526} C_VEL
LIN {X 0,Y 348.078,Z 279.755,A -85,B 0,C 180,E1 -13673.043,E2 -13673.043} C_VEL
LIN {X 0,Y 348.195,Z 279.735,A -85,B 0,C 180,E1 -13677.687,E2 -13677.687} C_VEL
LIN {X 0,Y 348.333,Z 279.717,A -85,B 0,C 180,E1 -13680.001,E2 -13680.001} C_VEL
LIN {X 0,Y 348.193,Z 279.735,A -85,B 0,C 180,E1 -13682.314,E2 -13682.314} C_VEL
LIN {X 0,Y 348.093,Z 279.753,A -85,B 0,C 180,E1 -13686.959,E2 -13686.959} C_VEL
LIN {X 0,Y 347.956,Z 279.766,A -85,B 0,C 180,E1 -13689.3,E2 -13689.3} C_VEL
LIN {X 0,Y 347.878,Z 279.778,A -85,B 0,C 180,E1 -13692.841,E2 -13692.841} C_VEL
LIN {X 0,Y 347.828,Z 279.781,A -85,B 0,C 180,E1 -13696.433,E2 -13696.433} C_VEL
LIN {X 0,Y 347.84,Z 279.784,A -85,B 0,C 180,E1 -13698.862,E2 -13698.862} C_VEL
LIN {X 0,Y 347.753,Z 279.792,A -85,B 0,C 180,E1 -13702.582,E2 -13702.582} C_VEL
LIN {X 0,Y 347.802,Z 279.787,A -85,B 0,C 180,E1 -13705.11,E2 -13705.11} C_VEL
LIN {X 0,Y 347.8,Z 279.783,A -85,B 0,C 180,E1 -13707.695,E2 -13707.695} C_VEL
LIN {X 0,Y 347.755,Z 279.79,A -85,B 0,C 180,E1 -13710.348,E2 -13710.348} C_VEL
LIN {X 0,Y 347.736,Z 279.794,A -85,B 0,C 180,E1 -13714.466,E2 -13714.466} C_VEL
LIN {X 0,Y 347.765,Z 279.788,A -85,B 0,C 180,E1 -13717.99,E2 -13717.99} C_VEL
LIN {X 0,Y 347.743,Z 279.79,A -85,B 0,C 180,E1 -13721.832,E2 -13721.832} C_VEL
LIN {X 0,Y 347.759,Z 279.792,A -85,B 0,C 180,E1 -13725.019,E2 -13725.019} C_VEL
LIN {X 0,Y 347.744,Z 279.793,A -85,B 0,C 180,E1 -13728.399,E2 -13728.399} C_VEL
LIN {X 0,Y 347.814,Z 279.92,A -85,B 0,C 180,E1 -13731.968,E2 -13731.968} C_VEL
LIN {X 0,Y 352.183,Z 297.191,A -85,B 0,C 180,E1 -13735.764,E2 -13735.764} C_VEL
LIN {X 0,Y 355.885,Z 312.722,A -85,B 0,C 180,E1 -13738.96,E2 -13738.96} C_VEL
LIN {X 0,Y 356.988,Z 317.019,A -85,B 0,C 180,E1 -13739.165,E2 -13739.165} C_VEL
LIN {X 0,Y 363.111,Z 357.822,A -85,B 0,C 180,E1 -13740.773,E2 -13740.773} C_VEL
LIN {X 0,Y 358.228,Z 479.415,A -85,B 0,C 180,E1 -13744.003,E2 -13744.003} C_VEL
LIN {X 0,Y 357.235,Z 495.024,A -85,B 0,C 180,E1 -13744.617,E2 -13744.617} C_VEL
LIN {X 0,Y 355.937,Z 511.215,A -85,B 0,C 180,E1 -13745.505,E2 -13745.505} C_VEL
LIN {X 0,Y 354.667,Z 525.262,A -85,B 0,C 180,E1 -13746.499,E2 -13746.499} C_VEL
LIN {X 0,Y 353.163,Z 539.816,A -85,B 0,C 180,E1 -13747.786,E2 -13747.786} C_VEL
LIN {X 0,Y 351.741,Z 553.132,A -85,B 0,C 180,E1 -13749.23,E2 -13749.23} C_VEL
LIN {X 0,Y 350.342,Z 565.333,A -85,B 0,C 180,E1 -13750.821,E2 -13750.821} C_VEL
LIN {X 0,Y 349.069,Z 577.44,A -85,B 0,C 180,E1 -13752.726,E2 -13752.726} C_VEL
LIN {X 0,Y 347.995,Z 588.216,A -85,B 0,C 180,E1 -13754.781,E2 -13754.781} C_VEL
LIN {X 0,Y 347.255,Z 596.331,A -85,B 0,C 180,E1 -13756.642,E2 -13756.642} C_VEL
LIN {X 0,Y 346.885,Z 602.544,A -85,B 0,C 180,E1 -13758.313,E2 -13758.313} C_VEL
LIN {X 0,Y 346.495,Z 609.656,A -85,B 0,C 180,E1 -13760.663,E2 -13760.663} C_VEL
LIN {X 0,Y 346.346,Z 615.137,A -85,B 0,C 180,E1 -13763.009,E2 -13763.009} C_VEL
LIN {X 0,Y 346.313,Z 619.122,A -85,B 0,C 180,E1 -13765.346,E2 -13765.346} C_VEL
LIN {X 0,Y 346.402,Z 621.704,A -85,B 0,C 180,E1 -13767.676,E2 -13767.676} C_VEL
LIN {X 0,Y 346.392,Z 622.901,A -85,B 0,C 180,E1 -13770.002,E2 -13770.002} C_VEL
LIN {X 0,Y 346.403,Z 623.001,A -85,B 0,C 180,E1 -13771.164,E2 -13771.164} C_VEL
LIN {X 0,Y 346.222,Z 622.204,A -85,B 0,C 180,E1 -13773.493,E2 -13773.493} C_VEL
LIN {X 0,Y 346.246,Z 619.962,A -85,B 0,C 180,E1 -13775.96,E2 -13775.96} C_VEL
LIN {X 0,Y 346.328,Z 616.731,A -85,B 0,C 180,E1 -13778.168,E2 -13778.168} C_VEL
LIN {X 0,Y 346.604,Z 611.983,A -85,B 0,C 180,E1 -13780.516,E2 -13780.516} C_VEL
LIN {X 0,Y 347.272,Z 605.784,A -85,B 0,C 180,E1 -13782.864,E2 -13782.864} C_VEL
LIN {X 0,Y 348.336,Z 598.012,A -85,B 0,C 180,E1 -13785.207,E2 -13785.207} C_VEL
LIN {X 0,Y 349.663,Z 589.78,A -85,B 0,C 180,E1 -13787.247,E2 -13787.247} C_VEL
LIN {X 0,Y 351.32,Z 579.986,A -85,B 0,C 180,E1 -13789.275,E2 -13789.275} C_VEL
LIN {X 0,Y 353.451,Z 568.315,A -85,B 0,C 180,E1 -13791.279,E2 -13791.279} C_VEL
LIN {X 0,Y 355.862,Z 555.423,A -85,B 0,C 180,E1 -13793.113,E2 -13793.113} C_VEL
LIN {X 0,Y 358.217,Z 542.527,A -85,B 0,C 180,E1 -13794.641,E2 -13794.641} C_VEL
LIN {X 0,Y 360.689,Z 528.577,A -85,B 0,C 180,E1 -13796.013,E2 -13796.013} C_VEL
LIN {X 0,Y 363.279,Z 513.688,A -85,B 0,C 180,E1 -13797.198,E2 -13797.198} C_VEL
LIN {X 0,Y 365.629,Z 498.435,A -85,B 0,C 180,E1 -13798.174,E2 -13798.174} C_VEL
LIN {X 0,Y 368.012,Z 480.971,A -85,B 0,C 180,E1 -13799.026,E2 -13799.026} C_VEL
LIN {X 0,Y 369.85,Z 462.49,A -85,B 0,C 180,E1 -13799.687,E2 -13799.687} C_VEL
LIN {X 0,Y 376.253,Z 394.365,A -85,B 0,C 180,E1 -13801.907,E2 -13801.907} C_VEL
LIN {X 0,Y 379.714,Z 361.521,A -85,B 0,C 180,E1 -13803.031,E2 -13803.031} C_VEL
LIN {X 0,Y 379.241,Z 349.895,A -85,B 0,C 180,E1 -13803.803,E2 -13803.803} C_VEL
LIN {X 0,Y 378.331,Z 338.632,A -85,B 0,C 180,E1 -13804.709,E2 -13804.709} C_VEL
LIN {X 0,Y 375.363,Z 330.8,A -85,B 0,C 180,E1 -13806.012,E2 -13806.012} C_VEL
LIN {X 0,Y 372.443,Z 324.465,A -85,B 0,C 180,E1 -13807.414,E2 -13807.414} C_VEL
LIN {X 0,Y 369.365,Z 318.069,A -85,B 0,C 180,E1 -13809.225,E2 -13809.225} C_VEL
LIN {X 0,Y 366.609,Z 312.855,A -85,B 0,C 180,E1 -13811.422,E2 -13811.422} C_VEL
LIN {X 0,Y 365.321,Z 309.799,A -85,B 0,C 180,E1 -13813.233,E2 -13813.233} C_VEL
LIN {X 0,Y 364.801,Z 308.151,A -85,B 0,C 180,E1 -13815.047,E2 -13815.047} C_VEL
LIN {X 0,Y 365.083,Z 308.02,A -85,B 0,C 180,E1 -13817.015,E2 -13817.015} C_VEL
LIN {X 0,Y 366.749,Z 309.367,A -85,B 0,C 180,E1 -13819.341,E2 -13819.341} C_VEL
LIN {X 0,Y 368.072,Z 310.414,A -85,B 0,C 180,E1 -13820.425,E2 -13820.425} C_VEL
LIN {X 0,Y 371.032,Z 313.981,A -85,B 0,C 180,E1 -13822.345,E2 -13822.345} C_VEL
LIN {X 0,Y 373.827,Z 317.839,A -85,B 0,C 180,E1 -13823.762,E2 -13823.762} C_VEL
LIN {X 0,Y 376.992,Z 322.635,A -85,B 0,C 180,E1 -13825.113,E2 -13825.113} C_VEL
LIN {X 0,Y 380.639,Z 328.915,A -85,B 0,C 180,E1 -13826.476,E2 -13826.476} C_VEL
LIN {X 0,Y 382.216,Z 332.371,A -85,B 0,C 180,E1 -13827.049,E2 -13827.049} C_VEL
LIN {X 0,Y 374.062,Z 404.607,A -85,B 0,C 180,E1 -13829.477,E2 -13829.477} C_VEL
LIN {X 0,Y 369.951,Z 449,A -85,B 0,C 180,E1 -13830.983,E2 -13830.983} C_VEL
LIN {X 0,Y 368.373,Z 463.676,A -85,B 0,C 180,E1 -13831.677,E2 -13831.677} C_VEL
LIN {X 0,Y 366.487,Z 478.531,A -85,B 0,C 180,E1 -13832.597,E2 -13832.597} C_VEL
LIN {X 0,Y 364.473,Z 492.367,A -85,B 0,C 180,E1 -13833.672,E2 -13833.672} C_VEL
LIN {X 0,Y 362.138,Z 506.611,A -85,B 0,C 180,E1 -13835.032,E2 -13835.032} C_VEL
LIN {X 0,Y 359.928,Z 518.976,A -85,B 0,C 180,E1 -13836.464,E2 -13836.464} C_VEL
LIN {X 0,Y 357.57,Z 530.655,A -85,B 0,C 180,E1 -13838.071,E2 -13838.071} C_VEL
LIN {X 0,Y 355.508,Z 540.859,A -85,B 0,C 180,E1 -13839.759,E2 -13839.759} C_VEL
LIN {X 0,Y 353.486,Z 550.87,A -85,B 0,C 180,E1 -13841.751,E2 -13841.751} C_VEL
LIN {X 0,Y 351.608,Z 559.239,A -85,B 0,C 180,E1 -13843.749,E2 -13843.749} C_VEL
LIN {X 0,Y 350.308,Z 565.301,A -85,B 0,C 180,E1 -13845.476,E2 -13845.476} C_VEL
LIN {X 0,Y 348.933,Z 571.883,A -85,B 0,C 180,E1 -13847.79,E2 -13847.79} C_VEL
LIN {X 0,Y 348.084,Z 576.961,A -85,B 0,C 180,E1 -13850.117,E2 -13850.117} C_VEL
LIN {X 0,Y 347.236,Z 580.95,A -85,B 0,C 180,E1 -13852.644,E2 -13852.644} C_VEL
LIN {X 0,Y 346.816,Z 582.623,A -85,B 0,C 180,E1 -13854.184,E2 -13854.184} C_VEL
LIN {X 0,Y 346.719,Z 584.117,A -85,B 0,C 180,E1 -13856.513,E2 -13856.513} C_VEL
LIN {X 0,Y 346.449,Z 584.404,A -85,B 0,C 180,E1 -13858.837,E2 -13858.837} C_VEL
LIN {X 0,Y 346.408,Z 583.437,A -85,B 0,C 180,E1 -13861.162,E2 -13861.162} C_VEL
LIN {X 0,Y 346.406,Z 581.197,A -85,B 0,C 180,E1 -13863.489,E2 -13863.489} C_VEL
LIN {X 0,Y 346.56,Z 577.642,A -85,B 0,C 180,E1 -13865.819,E2 -13865.819} C_VEL
LIN {X 0,Y 346.815,Z 572.704,A -85,B 0,C 180,E1 -13868.154,E2 -13868.154} C_VEL
LIN {X 0,Y 347.272,Z 566.262,A -85,B 0,C 180,E1 -13870.493,E2 -13870.493} C_VEL
LIN {X 0,Y 347.966,Z 559.217,A -85,B 0,C 180,E1 -13872.539,E2 -13872.539} C_VEL
LIN {X 0,Y 348.791,Z 550.119,A -85,B 0,C 180,E1 -13874.716,E2 -13874.716} C_VEL
LIN {X 0,Y 349.833,Z 540.415,A -85,B 0,C 180,E1 -13876.634,E2 -13876.634} C_VEL
LIN {X 0,Y 350.961,Z 529.878,A -85,B 0,C 180,E1 -13878.383,E2 -13878.383} C_VEL
LIN {X 0,Y 352.068,Z 519.563,A -85,B 0,C 180,E1 -13879.836,E2 -13879.836} C_VEL
LIN {X 0,Y 353.432,Z 506.145,A -85,B 0,C 180,E1 -13881.43,E2 -13881.43} C_VEL
LIN {X 0,Y 354.762,Z 492.923,A -85,B 0,C 180,E1 -13882.724,E2 -13882.724} C_VEL
LIN {X 0,Y 356.015,Z 478.588,A -85,B 0,C 180,E1 -13883.87,E2 -13883.87} C_VEL
LIN {X 0,Y 357.093,Z 464.588,A -85,B 0,C 180,E1 -13884.763,E2 -13884.763} C_VEL
LIN {X 0,Y 357.949,Z 449.161,A -85,B 0,C 180,E1 -13885.526,E2 -13885.526} C_VEL
LIN {X 0,Y 358.695,Z 433.204,A -85,B 0,C 180,E1 -13886.079,E2 -13886.079} C_VEL
LIN {X 0,Y 363.392,Z 315.844,A -85,B 0,C 180,E1 -13889.154,E2 -13889.154} C_VEL
LIN {X 0,Y 347.834,Z 280.192,A -85,B 0,C 180,E1 -13891.301,E2 -13891.301} C_VEL
LIN {X 0,Y 347.775,Z 279.792,A -85,B 0,C 180,E1 -13891.372,E2 -13891.372} C_VEL
LIN {X 0,Y 347.745,Z 279.791,A -85,B 0,C 180,E1 -13894.462,E2 -13894.462} C_VEL
LIN {X 0,Y 347.764,Z 279.793,A -85,B 0,C 180,E1 -13897.985,E2 -13897.985} C_VEL
LIN {X 0,Y 347.747,Z 279.796,A -85,B 0,C 180,E1 -13901.829,E2 -13901.829} C_VEL
LIN {X 0,Y 347.704,Z 279.795,A -85,B 0,C 180,E1 -13905.025,E2 -13905.025} C_VEL
LIN {X 0,Y 347.749,Z 279.79,A -85,B 0,C 180,E1 -13908.396,E2 -13908.396} C_VEL
LIN {X 0,Y 347.771,Z 279.79,A -85,B 0,C 180,E1 -13912.01,E2 -13912.01} C_VEL
LIN {X 0,Y 347.742,Z 279.794,A -85,B 0,C 180,E1 -13915.534,E2 -13915.534} C_VEL
LIN {X 0,Y 347.741,Z 279.792,A -85,B 0,C 180,E1 -13918.299,E2 -13918.299} C_VEL
LIN {X 0,Y 347.742,Z 279.791,A -85,B 0,C 180,E1 -13920.983,E2 -13920.983} C_VEL
LIN {X 0,Y 347.752,Z 279.794,A -85,B 0,C 180,E1 -13923.6,E2 -13923.6} C_VEL
LIN {X 0,Y 347.766,Z 279.789,A -85,B 0,C 180,E1 -13926.159,E2 -13926.159} C_VEL
LIN {X 0,Y 347.795,Z 279.787,A -85,B 0,C 180,E1 -13929.907,E2 -13929.907} C_VEL
LIN {X 0,Y 347.827,Z 279.785,A -85,B 0,C 180,E1 -13933.567,E2 -13933.567} C_VEL
LIN {X 0,Y 347.884,Z 279.774,A -85,B 0,C 180,E1 -13937.159,E2 -13937.159} C_VEL
LIN {X 0,Y 348.088,Z 279.754,A -85,B 0,C 180,E1 -13941.611,E2 -13941.611} C_VEL
LIN {X 0,Y 348.058,Z 279.752,A -85,B 0,C 180,E1 -13944.204,E2 -13944.204} C_VEL
LIN {X 0,Y 348.197,Z 279.739,A -85,B 0,C 180,E1 -13947.685,E2 -13947.685} C_VEL
LIN {X 0,Y 348.338,Z 279.718,A -85,B 0,C 180,E1 -13949.998,E2 -13949.998} C_VEL
LIN {X 0,Y 348.197,Z 279.734,A -85,B 0,C 180,E1 -13952.312,E2 -13952.312} C_VEL
LIN {X 0,Y 348.096,Z 279.747,A -85,B 0,C 180,E1 -13956.956,E2 -13956.956} C_VEL
LIN {X 0,Y 347.958,Z 279.767,A -85,B 0,C 180,E1 -13959.297,E2 -13959.297} C_VEL
LIN {X 0,Y 347.88,Z 279.774,A -85,B 0,C 180,E1 -13962.838,E2 -13962.838} C_VEL
LIN {X 0,Y 347.828,Z 279.779,A -85,B 0,C 180,E1 -13966.43,E2 -13966.43} C_VEL
LIN {X 0,Y 347.84,Z 279.779,A -85,B 0,C 180,E1 -13968.859,E2 -13968.859} C_VEL
LIN {X 0,Y 347.764,Z 279.788,A -85,B 0,C 180,E1 -13972.578,E2 -13972.578} C_VEL
LIN {X 0,Y 347.8,Z 279.786,A -85,B 0,C 180,E1 -13975.107,E2 -13975.107} C_VEL
LIN {X 0,Y 347.796,Z 279.787,A -85,B 0,C 180,E1 -13977.693,E2 -13977.693} C_VEL
LIN {X 0,Y 347.711,Z 279.792,A -85,B 0,C 180,E1 -13980.905,E2 -13980.905} C_VEL
LIN {X 0,Y 347.731,Z 279.792,A -85,B 0,C 180,E1 -13984.463,E2 -13984.463} C_VEL
LIN {X 0,Y 347.77,Z 279.788,A -85,B 0,C 180,E1 -13985.938,E2 -13985.938} C_VEL
LIN {X 0,Y 347.037,Z 279.882,A -85,B 0,C 180,E1 -13986.904,E2 -13986.904} C_VEL
LIN {X 0,Y 344.143,Z 280.239,A -85,B 0,C 180,E1 -13988.474,E2 -13988.474} C_VEL
LIN {X 0,Y 341.742,Z 280.54,A -85,B 0,C 180,E1 -13989.745,E2 -13989.745} C_VEL
LIN {X 0,Y 340.735,Z 280.665,A -85,B 0,C 180,E1 -13990.729,E2 -13990.729} C_VEL
LIN {X 0,Y 340.663,Z 280.676,A -85,B 0,C 180,E1 -13991.062,E2 -13991.062} C_VEL
LIN {X 0,Y 340.669,Z 280.672,A -85,B 0,C 180,E1 -13994.538,E2 -13994.538} C_VEL
LIN {X 0,Y 340.685,Z 280.67,A -85,B 0,C 180,E1 -13997.954,E2 -13997.954} C_VEL
LIN {X 0,Y 340.718,Z 280.667,A -85,B 0,C 180,E1 -14001.772,E2 -14001.772} C_VEL
LIN {X 0,Y 340.708,Z 280.669,A -85,B 0,C 180,E1 -14005.595,E2 -14005.595} C_VEL
LIN {X 0,Y 340.689,Z 280.672,A -85,B 0,C 180,E1 -14008.956,E2 -14008.956} C_VEL
LIN {X 0,Y 340.763,Z 280.66,A -85,B 0,C 180,E1 -14012.475,E2 -14012.475} C_VEL
LIN {X 0,Y 340.74,Z 280.664,A -85,B 0,C 180,E1 -14015.638,E2 -14015.638} C_VEL
LIN {X 0,Y 340.72,Z 280.668,A -85,B 0,C 180,E1 -14019.474,E2 -14019.474} C_VEL
LIN {X 0,Y 340.844,Z 280.65,A -85,B 0,C 180,E1 -14021.985,E2 -14021.985} C_VEL
LIN {X 0,Y 340.856,Z 280.649,A -85,B 0,C 180,E1 -14025.706,E2 -14025.706} C_VEL
LIN {X 0,Y 340.857,Z 280.652,A -85,B 0,C 180,E1 -14029.307,E2 -14029.307} C_VEL
LIN {X 0,Y 341.046,Z 280.629,A -85,B 0,C 180,E1 -14032.899,E2 -14032.899} C_VEL
LIN {X 0,Y 341.156,Z 280.612,A -85,B 0,C 180,E1 -14037.64,E2 -14037.64} C_VEL
LIN {X 0,Y 341.284,Z 280.595,A -85,B 0,C 180,E1 -14040.001,E2 -14040.001} C_VEL
LIN {X 0,Y 341.155,Z 280.612,A -85,B 0,C 180,E1 -14042.362,E2 -14042.362} C_VEL
LIN {X 0,Y 341.062,Z 280.627,A -85,B 0,C 180,E1 -14047.103,E2 -14047.103} C_VEL
LIN {X 0,Y 340.859,Z 280.651,A -85,B 0,C 180,E1 -14050.695,E2 -14050.695} C_VEL
LIN {X 0,Y 340.852,Z 280.65,A -85,B 0,C 180,E1 -14054.326,E2 -14054.326} C_VEL
LIN {X 0,Y 340.826,Z 280.654,A -85,B 0,C 180,E1 -14058.468,E2 -14058.468} C_VEL
LIN {X 0,Y 340.708,Z 280.667,A -85,B 0,C 180,E1 -14061.843,E2 -14061.843} C_VEL
LIN {X 0,Y 340.762,Z 280.66,A -85,B 0,C 180,E1 -14065.666,E2 -14065.666} C_VEL
LIN {X 0,Y 340.731,Z 280.665,A -85,B 0,C 180,E1 -14068.321,E2 -14068.321} C_VEL
LIN {X 0,Y 340.695,Z 280.672,A -85,B 0,C 180,E1 -14071.046,E2 -14071.046} C_VEL
LIN {X 0,Y 340.71,Z 280.668,A -85,B 0,C 180,E1 -14075.281,E2 -14075.281} C_VEL
LIN {X 0,Y 340.702,Z 280.67,A -85,B 0,C 180,E1 -14078.388,E2 -14078.388} C_VEL
LIN {X 0,Y 340.692,Z 280.669,A -85,B 0,C 180,E1 -14082.047,E2 -14082.047} C_VEL
LIN {X 0,Y 340.676,Z 280.671,A -85,B 0,C 180,E1 -14085.463,E2 -14085.463} C_VEL
LIN {X 0,Y 340.68,Z 280.676,A -85,B 0,C 180,E1 -14088.692,E2 -14088.692} C_VEL
LIN {X 0,Y 340.73,Z 280.754,A -85,B 0,C 180,E1 -14091.53,E2 -14091.53} C_VEL
LIN {X 0,Y 345.388,Z 299.07,A -85,B 0,C 180,E1 -14095.641,E2 -14095.641} C_VEL
LIN {X 0,Y 348.492,Z 312.234,A -85,B 0,C 180,E1 -14098.423,E2 -14098.423} C_VEL
LIN {X 0,Y 350.449,Z 317.918,A -85,B 0,C 180,E1 -14098.739,E2 -14098.739} C_VEL
LIN {X 0,Y 356.486,Z 359.057,A -85,B 0,C 180,E1 -14100.393,E2 -14100.393} C_VEL
LIN {X 0,Y 351.455,Z 478.854,A -85,B 0,C 180,E1 -14103.663,E2 -14103.663} C_VEL
LIN {X 0,Y 350.438,Z 494.627,A -85,B 0,C 180,E1 -14104.298,E2 -14104.298} C_VEL
LIN {X 0,Y 349.13,Z 510.071,A -85,B 0,C 180,E1 -14105.154,E2 -14105.154} C_VEL
LIN {X 0,Y 347.838,Z 524.246,A -85,B 0,C 180,E1 -14106.168,E2 -14106.168} C_VEL
LIN {X 0,Y 346.295,Z 538.899,A -85,B 0,C 180,E1 -14107.478,E2 -14107.478} C_VEL
LIN {X 0,Y 344.802,Z 552.29,A -85,B 0,C 180,E1 -14108.948,E2 -14108.948} C_VEL
LIN {X 0,Y 343.42,Z 564.164,A -85,B 0,C 180,E1 -14110.512,E2 -14110.512} C_VEL
LIN {X 0,Y 342.346,Z 574.186,A -85,B 0,C 180,E1 -14112.067,E2 -14112.067} C_VEL
LIN {X 0,Y 341.301,Z 583.97,A -85,B 0,C 180,E1 -14113.862,E2 -14113.862} C_VEL
LIN {X 0,Y 340.43,Z 593.718,A -85,B 0,C 180,E1 -14116,E2 -14116} C_VEL
LIN {X 0,Y 339.855,Z 601.468,A -85,B 0,C 180,E1 -14118.067,E2 -14118.067} C_VEL
LIN {X 0,Y 339.414,Z 608.747,A -85,B 0,C 180,E1 -14120.467,E2 -14120.467} C_VEL
LIN {X 0,Y 339.288,Z 614.36,A -85,B 0,C 180,E1 -14122.862,E2 -14122.862} C_VEL
LIN {X 0,Y 339.298,Z 616.593,A -85,B 0,C 180,E1 -14124.057,E2 -14124.057} C_VEL
LIN {X 0,Y 339.186,Z 619.942,A -85,B 0,C 180,E1 -14126.438,E2 -14126.438} C_VEL
LIN {X 0,Y 339.324,Z 621.103,A -85,B 0,C 180,E1 -14127.628,E2 -14127.628} C_VEL
LIN {X 0,Y 339.33,Z 622.388,A -85,B 0,C 180,E1 -14130.002,E2 -14130.002} C_VEL
LIN {X 0,Y 339.339,Z 622.534,A -85,B 0,C 180,E1 -14131.188,E2 -14131.188} C_VEL
LIN {X 0,Y 339.142,Z 621.826,A -85,B 0,C 180,E1 -14133.566,E2 -14133.566} C_VEL
LIN {X 0,Y 339.172,Z 619.832,A -85,B 0,C 180,E1 -14135.948,E2 -14135.948} C_VEL
LIN {X 0,Y 339.253,Z 616.535,A -85,B 0,C 180,E1 -14138.34,E2 -14138.34} C_VEL
LIN {X 0,Y 339.565,Z 611.891,A -85,B 0,C 180,E1 -14140.737,E2 -14140.737} C_VEL
LIN {X 0,Y 340.282,Z 605.815,A -85,B 0,C 180,E1 -14143.133,E2 -14143.133} C_VEL
LIN {X 0,Y 341.451,Z 598.176,A -85,B 0,C 180,E1 -14145.522,E2 -14145.522} C_VEL
LIN {X 0,Y 343.079,Z 588.788,A -85,B 0,C 180,E1 -14147.897,E2 -14147.897} C_VEL
LIN {X 0,Y 344.901,Z 578.944,A -85,B 0,C 180,E1 -14149.958,E2 -14149.958} C_VEL
LIN {X 0,Y 347.264,Z 567.233,A -85,B 0,C 180,E1 -14151.989,E2 -14151.989} C_VEL
LIN {X 0,Y 349.829,Z 554.332,A -85,B 0,C 180,E1 -14153.849,E2 -14153.849} C_VEL
LIN {X 0,Y 352.675,Z 540.155,A -85,B 0,C 180,E1 -14155.528,E2 -14155.528} C_VEL
LIN {X 0,Y 355.377,Z 525.816,A -85,B 0,C 180,E1 -14156.926,E2 -14156.926} C_VEL
LIN {X 0,Y 358.081,Z 510.866,A -85,B 0,C 180,E1 -14158.104,E2 -14158.104} C_VEL
LIN {X 0,Y 360.501,Z 496.435,A -85,B 0,C 180,E1 -14159.01,E2 -14159.01} C_VEL
LIN {X 0,Y 363.016,Z 478.853,A -85,B 0,C 180,E1 -14159.864,E2 -14159.864} C_VEL
LIN {X 0,Y 365.362,Z 455.718,A -85,B 0,C 180,E1 -14160.688,E2 -14160.688} C_VEL
LIN {X 0,Y 372.185,Z 390.481,A -85,B 0,C 180,E1 -14162.882,E2 -14162.882} C_VEL
LIN {X 0,Y 375.342,Z 362.892,A -85,B 0,C 180,E1 -14163.856,E2 -14163.856} C_VEL
LIN {X 0,Y 374.97,Z 350.653,A -85,B 0,C 180,E1 -14164.724,E2 -14164.724} C_VEL
LIN {X 0,Y 374.389,Z 342.56,A -85,B 0,C 180,E1 -14165.419,E2 -14165.419} C_VEL
LIN {X 0,Y 371.638,Z 335.1,A -85,B 0,C 180,E1 -14166.76,E2 -14166.76} C_VEL
LIN {X 0,Y 369.536,Z 330.189,A -85,B 0,C 180,E1 -14167.889,E2 -14167.889} C_VEL
LIN {X 0,Y 366.88,Z 324.236,A -85,B 0,C 180,E1 -14169.614,E2 -14169.614} C_VEL
LIN {X 0,Y 364.413,Z 319.098,A -85,B 0,C 180,E1 -14171.854,E2 -14171.854} C_VEL
LIN {X 0,Y 363.351,Z 316.12,A -85,B 0,C 180,E1 -14173.725,E2 -14173.725} C_VEL
LIN {X 0,Y 363.027,Z 314.925,A -85,B 0,C 180,E1 -14175.372,E2 -14175.372} C_VEL
LIN {X 0,Y 363.58,Z 315.12,A -85,B 0,C 180,E1 -14177.569,E2 -14177.569} C_VEL
LIN {X 0,Y 365.885,Z 316.831,A -85,B 0,C 180,E1 -14180.098,E2 -14180.098} C_VEL
LIN {X 0,Y 368.738,Z 320.514,A -85,B 0,C 180,E1 -14182.096,E2 -14182.096} C_VEL
LIN {X 0,Y 371.31,Z 324.226,A -85,B 0,C 180,E1 -14183.478,E2 -14183.478} C_VEL
LIN {X 0,Y 374.561,Z 329.362,A -85,B 0,C 180,E1 -14184.94,E2 -14184.94} C_VEL
LIN {X 0,Y 377.809,Z 335.546,A -85,B 0,C 180,E1 -14186.24,E2 -14186.24} C_VEL
LIN {X 0,Y 368.938,Z 409.394,A -85,B 0,C 180,E1 -14188.808,E2 -14188.808} C_VEL
LIN {X 0,Y 364.878,Z 449.699,A -85,B 0,C 180,E1 -14190.216,E2 -14190.216} C_VEL
LIN {X 0,Y 363.113,Z 464.792,A -85,B 0,C 180,E1 -14190.954,E2 -14190.954} C_VEL
LIN {X 0,Y 360.901,Z 480.706,A -85,B 0,C 180,E1 -14191.978,E2 -14191.978} C_VEL
LIN {X 0,Y 358.782,Z 494.104,A -85,B 0,C 180,E1 -14193.064,E2 -14193.064} C_VEL
LIN {X 0,Y 356.287,Z 508.06,A -85,B 0,C 180,E1 -14194.437,E2 -14194.437} C_VEL
LIN {X 0,Y 353.888,Z 520.436,A -85,B 0,C 180,E1 -14195.915,E2 -14195.915} C_VEL
LIN {X 0,Y 351.246,Z 532.631,A -85,B 0,C 180,E1 -14197.655,E2 -14197.655} C_VEL
LIN {X 0,Y 349.062,Z 542.565,A -85,B 0,C 180,E1 -14199.368,E2 -14199.368} C_VEL
LIN {X 0,Y 346.899,Z 552.349,A -85,B 0,C 180,E1 -14201.391,E2 -14201.391} C_VEL
LIN {X 0,Y 344.729,Z 561.371,A -85,B 0,C 180,E1 -14203.652,E2 -14203.652} C_VEL
LIN {X 0,Y 343.2,Z 568.166,A -85,B 0,C 180,E1 -14205.774,E2 -14205.774} C_VEL
LIN {X 0,Y 341.793,Z 574.231,A -85,B 0,C 180,E1 -14208.133,E2 -14208.133} C_VEL
LIN {X 0,Y 340.896,Z 578.826,A -85,B 0,C 180,E1 -14210.506,E2 -14210.506} C_VEL
LIN {X 0,Y 340.152,Z 582.103,A -85,B 0,C 180,E1 -14212.878,E2 -14212.878} C_VEL
LIN {X 0,Y 339.667,Z 584.121,A -85,B 0,C 180,E1 -14215.252,E2 -14215.252} C_VEL
LIN {X 0,Y 339.529,Z 584.892,A -85,B 0,C 180,E1 -14217.626,E2 -14217.626} C_VEL
LIN {X 0,Y 339.317,Z 584.441,A -85,B 0,C 180,E1 -14219.999,E2 -14219.999} C_VEL
LIN {X 0,Y 339.326,Z 582.738,A -85,B 0,C 180,E1 -14222.373,E2 -14222.373} C_VEL
LIN {X 0,Y 339.412,Z 579.749,A -85,B 0,C 180,E1 -14224.75,E2 -14224.75} C_VEL
LIN {X 0,Y 339.609,Z 575.395,A -85,B 0,C 180,E1 -14227.132,E2 -14227.132} C_VEL
LIN {X 0,Y 339.968,Z 569.585,A -85,B 0,C 180,E1 -14229.518,E2 -14229.518} C_VEL
LIN {X 0,Y 340.577,Z 562.145,A -85,B 0,C 180,E1 -14231.908,E2 -14231.908} C_VEL
LIN {X 0,Y 341.444,Z 554.143,A -85,B 0,C 180,E1 -14233.995,E2 -14233.995} C_VEL
LIN {X 0,Y 342.398,Z 544.452,A -85,B 0,C 180,E1 -14236.086,E2 -14236.086} C_VEL
LIN {X 0,Y 343.52,Z 534.579,A -85,B 0,C 180,E1 -14237.87,E2 -14237.87} C_VEL
LIN {X 0,Y 344.892,Z 522.863,A -85,B 0,C 180,E1 -14239.646,E2 -14239.646} C_VEL
LIN {X 0,Y 346.132,Z 510.708,A -85,B 0,C 180,E1 -14241.194,E2 -14241.194} C_VEL
LIN {X 0,Y 347.479,Z 497.449,A -85,B 0,C 180,E1 -14242.598,E2 -14242.598} C_VEL
LIN {X 0,Y 348.722,Z 484.038,A -85,B 0,C 180,E1 -14243.769,E2 -14243.769} C_VEL
LIN {X 0,Y 349.991,Z 468.383,A -85,B 0,C 180,E1 -14244.861,E2 -14244.861} C_VEL
LIN {X 0,Y 351.028,Z 451.976,A -85,B 0,C 180,E1 -14245.731,E2 -14245.731} C_VEL
LIN {X 0,Y 351.827,Z 436.827,A -85,B 0,C 180,E1 -14246.308,E2 -14246.308} C_VEL
LIN {X 0,Y 356.693,Z 317.382,A -85,B 0,C 180,E1 -14249.55,E2 -14249.55} C_VEL
LIN {X 0,Y 340.797,Z 281.232,A -85,B 0,C 180,E1 -14251.791,E2 -14251.791} C_VEL
LIN {X 0,Y 340.723,Z 280.671,A -85,B 0,C 180,E1 -14251.824,E2 -14251.824} C_VEL
LIN {X 0,Y 340.718,Z 280.666,A -85,B 0,C 180,E1 -14255.277,E2 -14255.277} C_VEL
LIN {X 0,Y 340.694,Z 280.67,A -85,B 0,C 180,E1 -14258.381,E2 -14258.381} C_VEL
LIN {X 0,Y 340.696,Z 280.672,A -85,B 0,C 180,E1 -14262.043,E2 -14262.043} C_VEL
LIN {X 0,Y 340.651,Z 280.676,A -85,B 0,C 180,E1 -14266.225,E2 -14266.225} C_VEL
LIN {X 0,Y 340.687,Z 280.675,A -85,B 0,C 180,E1 -14269.751,E2 -14269.751} C_VEL
LIN {X 0,Y 340.702,Z 280.669,A -85,B 0,C 180,E1 -14273.257,E2 -14273.257} C_VEL
LIN {X 0,Y 340.69,Z 280.671,A -85,B 0,C 180,E1 -14276.152,E2 -14276.152} C_VEL
LIN {X 0,Y 340.718,Z 280.668,A -85,B 0,C 180,E1 -14280.033,E2 -14280.033} C_VEL
LIN {X 0,Y 340.719,Z 280.666,A -85,B 0,C 180,E1 -14283.011,E2 -14283.011} C_VEL
LIN {X 0,Y 340.738,Z 280.668,A -85,B 0,C 180,E1 -14285.636,E2 -14285.636} C_VEL
LIN {X 0,Y 340.725,Z 280.668,A -85,B 0,C 180,E1 -14289.471,E2 -14289.471} C_VEL
LIN {X 0,Y 340.787,Z 280.66,A -85,B 0,C 180,E1 -14291.979,E2 -14291.979} C_VEL
LIN {X 0,Y 340.864,Z 280.653,A -85,B 0,C 180,E1 -14295.703,E2 -14295.703} C_VEL
LIN {X 0,Y 340.864,Z 280.65,A -85,B 0,C 180,E1 -14299.304,E2 -14299.304} C_VEL
LIN {X 0,Y 341.067,Z 280.622,A -85,B 0,C 180,E1 -14302.896,E2 -14302.896} C_VEL
LIN {X 0,Y 341.159,Z 280.616,A -85,B 0,C 180,E1 -14307.637,E2 -14307.637} C_VEL
LIN {X 0,Y 341.288,Z 280.596,A -85,B 0,C 180,E1 -14309.998,E2 -14309.998} C_VEL
LIN {X 0,Y 341.159,Z 280.61,A -85,B 0,C 180,E1 -14312.36,E2 -14312.36} C_VEL
LIN {X 0,Y 341.065,Z 280.624,A -85,B 0,C 180,E1 -14317.1,E2 -14317.1} C_VEL
LIN {X 0,Y 340.861,Z 280.648,A -85,B 0,C 180,E1 -14320.692,E2 -14320.692} C_VEL
LIN {X 0,Y 340.853,Z 280.649,A -85,B 0,C 180,E1 -14324.323,E2 -14324.323} C_VEL
LIN {X 0,Y 340.826,Z 280.652,A -85,B 0,C 180,E1 -14328.465,E2 -14328.465} C_VEL
LIN {X 0,Y 340.742,Z 280.664,A -85,B 0,C 180,E1 -14331.856,E2 -14331.856} C_VEL
LIN {X 0,Y 340.76,Z 280.663,A -85,B 0,C 180,E1 -14335.663,E2 -14335.663} C_VEL
LIN {X 0,Y 340.716,Z 280.666,A -85,B 0,C 180,E1 -14338.32,E2 -14338.32} C_VEL
LIN {X 0,Y 340.685,Z 280.672,A -85,B 0,C 180,E1 -14341.044,E2 -14341.044} C_VEL
LIN {X 0,Y 340.705,Z 280.672,A -85,B 0,C 180,E1 -14345.278,E2 -14345.278} C_VEL
LIN {X 0,Y 340.698,Z 280.668,A -85,B 0,C 180,E1 -14348.386,E2 -14348.386} C_VEL
LIN {X 0,Y 340.663,Z 280.676,A -85,B 0,C 180,E1 -14351.062,E2 -14351.062} C_VEL
LIN {X 0,Y 340.022,Z 280.762,A -85,B 0,C 180,E1 -14352.049,E2 -14352.049} C_VEL
LIN {X 0,Y 337.178,Z 281.117,A -85,B 0,C 180,E1 -14353.654,E2 -14353.654} C_VEL
LIN {X 0,Y 334.742,Z 281.415,A -85,B 0,C 180,E1 -14354.954,E2 -14354.954} C_VEL
LIN {X 0,Y 333.682,Z 281.542,A -85,B 0,C 180,E1 -14355.96,E2 -14355.96} C_VEL
LIN {X 0,Y 333.589,Z 281.552,A -85,B 0,C 180,E1 -14356.301,E2 -14356.301} C_VEL
LIN {X 0,Y 333.633,Z 281.553,A -85,B 0,C 180,E1 -14359.315,E2 -14359.315} C_VEL
LIN {X 0,Y 333.651,Z 281.551,A -85,B 0,C 180,E1 -14363.168,E2 -14363.168} C_VEL
LIN {X 0,Y 333.66,Z 281.549,A -85,B 0,C 180,E1 -14365.341,E2 -14365.341} C_VEL
LIN {X 0,Y 333.688,Z 281.542,A -85,B 0,C 180,E1 -14369.71,E2 -14369.71} C_VEL
LIN {X 0,Y 333.728,Z 281.536,A -85,B 0,C 180,E1 -14372.401,E2 -14372.401} C_VEL
LIN {X 0,Y 333.712,Z 281.543,A -85,B 0,C 180,E1 -14375.091,E2 -14375.091} C_VEL
LIN {X 0,Y 333.66,Z 281.549,A -85,B 0,C 180,E1 -14379.019,E2 -14379.019} C_VEL
LIN {X 0,Y 333.779,Z 281.531,A -85,B 0,C 180,E1 -14381.59,E2 -14381.59} C_VEL
LIN {X 0,Y 333.795,Z 281.529,A -85,B 0,C 180,E1 -14385.577,E2 -14385.577} C_VEL
LIN {X 0,Y 333.82,Z 281.531,A -85,B 0,C 180,E1 -14389.079,E2 -14389.079} C_VEL
LIN {X 0,Y 333.999,Z 281.505,A -85,B 0,C 180,E1 -14392.748,E2 -14392.748} C_VEL
LIN {X 0,Y 333.795,Z 281.532,A -85,B 0,C 180,E1 -14395.17,E2 -14395.17} C_VEL
LIN {X 0,Y 334.094,Z 281.492,A -85,B 0,C 180,E1 -14397.59,E2 -14397.59} C_VEL
LIN {X 0,Y 334.235,Z 281.473,A -85,B 0,C 180,E1 -14400.001,E2 -14400.001} C_VEL
LIN {X 0,Y 334.092,Z 281.492,A -85,B 0,C 180,E1 -14402.412,E2 -14402.412} C_VEL
LIN {X 0,Y 334.012,Z 281.504,A -85,B 0,C 180,E1 -14407.254,E2 -14407.254} C_VEL
LIN {X 0,Y 333.822,Z 281.53,A -85,B 0,C 180,E1 -14410.923,E2 -14410.923} C_VEL
LIN {X 0,Y 333.797,Z 281.53,A -85,B 0,C 180,E1 -14414.636,E2 -14414.636} C_VEL
LIN {X 0,Y 333.785,Z 281.532,A -85,B 0,C 180,E1 -14418.656,E2 -14418.656} C_VEL
LIN {X 0,Y 333.646,Z 281.547,A -85,B 0,C 180,E1 -14422.282,E2 -14422.282} C_VEL
LIN {X 0,Y 333.725,Z 281.537,A -85,B 0,C 180,E1 -14426.248,E2 -14426.248} C_VEL
LIN {X 0,Y 333.701,Z 281.544,A -85,B 0,C 180,E1 -14428.974,E2 -14428.974} C_VEL
LIN {X 0,Y 333.635,Z 281.551,A -85,B 0,C 180,E1 -14432.589,E2 -14432.589} C_VEL
LIN {X 0,Y 333.668,Z 281.544,A -85,B 0,C 180,E1 -14436.141,E2 -14436.141} C_VEL
LIN {X 0,Y 333.639,Z 281.549,A -85,B 0,C 180,E1 -14439.194,E2 -14439.194} C_VEL
LIN {X 0,Y 333.627,Z 281.552,A -85,B 0,C 180,E1 -14442.502,E2 -14442.502} C_VEL
LIN {X 0,Y 333.613,Z 281.551,A -85,B 0,C 180,E1 -14445.961,E2 -14445.961} C_VEL
LIN {X 0,Y 333.642,Z 281.551,A -85,B 0,C 180,E1 -14449.317,E2 -14449.317} C_VEL
LIN {X 0,Y 333.704,Z 281.724,A -85,B 0,C 180,E1 -14451.126,E2 -14451.126} C_VEL
LIN {X 0,Y 338.153,Z 299.293,A -85,B 0,C 180,E1 -14455.157,E2 -14455.157} C_VEL
LIN {X 0,Y 341.211,Z 312.142,A -85,B 0,C 180,E1 -14457.894,E2 -14457.894} C_VEL
LIN {X 0,Y 344.075,Z 320.077,A -85,B 0,C 180,E1 -14458.355,E2 -14458.355} C_VEL
LIN {X 0,Y 349.818,Z 360.46,A -85,B 0,C 180,E1 -14460.011,E2 -14460.011} C_VEL
LIN {X 0,Y 344.626,Z 479.008,A -85,B 0,C 180,E1 -14463.345,E2 -14463.345} C_VEL
LIN {X 0,Y 343.591,Z 494.598,A -85,B 0,C 180,E1 -14463.995,E2 -14463.995} C_VEL
LIN {X 0,Y 342.261,Z 509.893,A -85,B 0,C 180,E1 -14464.864,E2 -14464.864} C_VEL
LIN {X 0,Y 340.854,Z 524.887,A -85,B 0,C 180,E1 -14465.972,E2 -14465.972} C_VEL
LIN {X 0,Y 339.276,Z 539.35,A -85,B 0,C 180,E1 -14467.308,E2 -14467.308} C_VEL
LIN {X 0,Y 337.76,Z 552.602,A -85,B 0,C 180,E1 -14468.808,E2 -14468.808} C_VEL
LIN {X 0,Y 336.233,Z 565.815,A -85,B 0,C 180,E1 -14470.623,E2 -14470.623} C_VEL
LIN {X 0,Y 334.901,Z 577.702,A -85,B 0,C 180,E1 -14472.602,E2 -14472.602} C_VEL
LIN {X 0,Y 333.95,Z 586.896,A -85,B 0,C 180,E1 -14474.437,E2 -14474.437} C_VEL
LIN {X 0,Y 333.096,Z 595.895,A -85,B 0,C 180,E1 -14476.582,E2 -14476.582} C_VEL
LIN {X 0,Y 332.689,Z 602.361,A -85,B 0,C 180,E1 -14478.425,E2 -14478.425} C_VEL
LIN {X 0,Y 332.316,Z 609.338,A -85,B 0,C 180,E1 -14480.875,E2 -14480.875} C_VEL
LIN {X 0,Y 332.224,Z 614.69,A -85,B 0,C 180,E1 -14483.321,E2 -14483.321} C_VEL
LIN {X 0,Y 332.192,Z 617.716,A -85,B 0,C 180,E1 -14485.147,E2 -14485.147} C_VEL
LIN {X 0,Y 332.232,Z 620.48,A -85,B 0,C 180,E1 -14487.577,E2 -14487.577} C_VEL
LIN {X 0,Y 332.294,Z 621.345,A -85,B 0,C 180,E1 -14488.79,E2 -14488.79} C_VEL
LIN {X 0,Y 332.276,Z 622.064,A -85,B 0,C 180,E1 -14491.214,E2 -14491.214} C_VEL
LIN {X 0,Y 332.064,Z 621.451,A -85,B 0,C 180,E1 -14493.642,E2 -14493.642} C_VEL
LIN {X 0,Y 332.073,Z 619.556,A -85,B 0,C 180,E1 -14496.076,E2 -14496.076} C_VEL
LIN {X 0,Y 332.19,Z 616.363,A -85,B 0,C 180,E1 -14498.518,E2 -14498.518} C_VEL
LIN {X 0,Y 332.53,Z 611.822,A -85,B 0,C 180,E1 -14500.967,E2 -14500.967} C_VEL
LIN {X 0,Y 333.31,Z 605.86,A -85,B 0,C 180,E1 -14503.413,E2 -14503.413} C_VEL
LIN {X 0,Y 334.571,Z 598.374,A -85,B 0,C 180,E1 -14505.849,E2 -14505.849} C_VEL
LIN {X 0,Y 336.309,Z 589.19,A -85,B 0,C 180,E1 -14508.27,E2 -14508.27} C_VEL
LIN {X 0,Y 338.238,Z 579.555,A -85,B 0,C 180,E1 -14510.369,E2 -14510.369} C_VEL
LIN {X 0,Y 340.762,Z 568.118,A -85,B 0,C 180,E1 -14512.431,E2 -14512.431} C_VEL
LIN {X 0,Y 343.461,Z 555.55,A -85,B 0,C 180,E1 -14514.32,E2 -14514.32} C_VEL
LIN {X 0,Y 346.418,Z 541.806,A -85,B 0,C 180,E1 -14516.024,E2 -14516.024} C_VEL
LIN {X 0,Y 349.185,Z 528.294,A -85,B 0,C 180,E1 -14517.413,E2 -14517.413} C_VEL
LIN {X 0,Y 352.394,Z 512.007,A -85,B 0,C 180,E1 -14518.761,E2 -14518.761} C_VEL
LIN {X 0,Y 354.907,Z 498.144,A -85,B 0,C 180,E1 -14519.675,E2 -14519.675} C_VEL
LIN {X 0,Y 357.664,Z 480.927,A -85,B 0,C 180,E1 -14520.561,E2 -14520.561} C_VEL
LIN {X 0,Y 359.836,Z 462.263,A -85,B 0,C 180,E1 -14521.294,E2 -14521.294} C_VEL
LIN {X 0,Y 366.761,Z 400.087,A -85,B 0,C 180,E1 -14523.431,E2 -14523.431} C_VEL
LIN {X 0,Y 371.181,Z 364.433,A -85,B 0,C 180,E1 -14524.71,E2 -14524.71} C_VEL
LIN {X 0,Y 370.984,Z 352.036,A -85,B 0,C 180,E1 -14525.633,E2 -14525.633} C_VEL
LIN {X 0,Y 370.697,Z 346.8,A -85,B 0,C 180,E1 -14526.108,E2 -14526.108} C_VEL
LIN {X 0,Y 368.536,Z 340.556,A -85,B 0,C 180,E1 -14527.283,E2 -14527.283} C_VEL
LIN {X 0,Y 366.753,Z 336.022,A -85,B 0,C 180,E1 -14528.348,E2 -14528.348} C_VEL
LIN {X 0,Y 364.488,Z 330.47,A -85,B 0,C 180,E1 -14529.989,E2 -14529.989} C_VEL
LIN {X 0,Y 362.277,Z 325.476,A -85,B 0,C 180,E1 -14532.238,E2 -14532.238} C_VEL
LIN {X 0,Y 361.461,Z 322.785,A -85,B 0,C 180,E1 -14533.994,E2 -14533.994} C_VEL
LIN {X 0,Y 361.262,Z 321.742,A -85,B 0,C 180,E1 -14535.545,E2 -14535.545} C_VEL
LIN {X 0,Y 361.809,Z 321.998,A -85,B 0,C 180,E1 -14537.574,E2 -14537.574} C_VEL
LIN {X 0,Y 363.881,Z 323.583,A -85,B 0,C 180,E1 -14539.941,E2 -14539.941} C_VEL
LIN {X 0,Y 366.66,Z 327.401,A -85,B 0,C 180,E1 -14541.983,E2 -14541.983} C_VEL
LIN {X 0,Y 368.943,Z 330.864,A -85,B 0,C 180,E1 -14543.267,E2 -14543.267} C_VEL
LIN {X 0,Y 371.912,Z 335.844,A -85,B 0,C 180,E1 -14544.678,E2 -14544.678} C_VEL
LIN {X 0,Y 373.66,Z 339.348,A -85,B 0,C 180,E1 -14545.443,E2 -14545.443} C_VEL
LIN {X 0,Y 364.21,Z 412.133,A -85,B 0,C 180,E1 -14548.031,E2 -14548.031} C_VEL
LIN {X 0,Y 359.996,Z 450.382,A -85,B 0,C 180,E1 -14549.407,E2 -14549.407} C_VEL
LIN {X 0,Y 358.152,Z 464.974,A -85,B 0,C 180,E1 -14550.137,E2 -14550.137} C_VEL
LIN {X 0,Y 355.986,Z 479.521,A -85,B 0,C 180,E1 -14551.073,E2 -14551.073} C_VEL
LIN {X 0,Y 353.689,Z 493.103,A -85,B 0,C 180,E1 -14552.162,E2 -14552.162} C_VEL
LIN {X 0,Y 350.777,Z 508.43,A -85,B 0,C 180,E1 -14553.686,E2 -14553.686} C_VEL
LIN {X 0,Y 348.118,Z 521.099,A -85,B 0,C 180,E1 -14555.224,E2 -14555.224} C_VEL
LIN {X 0,Y 345.287,Z 533.196,A -85,B 0,C 180,E1 -14556.982,E2 -14556.982} C_VEL
LIN {X 0,Y 342.972,Z 542.834,A -85,B 0,C 180,E1 -14558.67,E2 -14558.67} C_VEL
LIN {X 0,Y 340.603,Z 552.622,A -85,B 0,C 180,E1 -14560.722,E2 -14560.722} C_VEL
LIN {X 0,Y 338.248,Z 561.883,A -85,B 0,C 180,E1 -14563.088,E2 -14563.088} C_VEL
LIN {X 0,Y 336.756,Z 567.607,A -85,B 0,C 180,E1 -14564.877,E2 -14564.877} C_VEL
LIN {X 0,Y 335.186,Z 573.879,A -85,B 0,C 180,E1 -14567.281,E2 -14567.281} C_VEL
LIN {X 0,Y 334.178,Z 578.676,A -85,B 0,C 180,E1 -14569.702,E2 -14569.702} C_VEL
LIN {X 0,Y 333.522,Z 581.42,A -85,B 0,C 180,E1 -14571.517,E2 -14571.517} C_VEL
LIN {X 0,Y 332.758,Z 583.945,A -85,B 0,C 180,E1 -14573.937,E2 -14573.937} C_VEL
LIN {X 0,Y 332.586,Z 585.197,A -85,B 0,C 180,E1 -14576.364,E2 -14576.364} C_VEL
LIN {X 0,Y 332.314,Z 585.243,A -85,B 0,C 180,E1 -14578.787,E2 -14578.787} C_VEL
LIN {X 0,Y 332.222,Z 584.042,A -85,B 0,C 180,E1 -14581.211,E2 -14581.211} C_VEL
LIN {X 0,Y 332.243,Z 581.58,A -85,B 0,C 180,E1 -14583.637,E2 -14583.637} C_VEL
LIN {X 0,Y 332.396,Z 577.791,A -85,B 0,C 180,E1 -14586.067,E2 -14586.067} C_VEL
LIN {X 0,Y 332.695,Z 572.587,A -85,B 0,C 180,E1 -14588.503,E2 -14588.503} C_VEL
LIN {X 0,Y 333.185,Z 565.827,A -85,B 0,C 180,E1 -14590.942,E2 -14590.942} C_VEL
LIN {X 0,Y 334.011,Z 558.504,A -85,B 0,C 180,E1 -14593.072,E2 -14593.072} C_VEL
LIN {X 0,Y 334.871,Z 549.133,A -85,B 0,C 180,E1 -14595.311,E2 -14595.311} C_VEL
LIN {X 0,Y 336.048,Z 538.878,A -85,B 0,C 180,E1 -14597.338,E2 -14597.338} C_VEL
LIN {X 0,Y 337.302,Z 527.887,A -85,B 0,C 180,E1 -14599.156,E2 -14599.156} C_VEL
LIN {X 0,Y 338.567,Z 516.189,A -85,B 0,C 180,E1 -14600.787,E2 -14600.787} C_VEL
LIN {X 0,Y 340.022,Z 502.981,A -85,B 0,C 180,E1 -14602.32,E2 -14602.32} C_VEL
LIN {X 0,Y 341.434,Z 488.913,A -85,B 0,C 180,E1 -14603.663,E2 -14603.663} C_VEL
LIN {X 0,Y 342.819,Z 473.412,A -85,B 0,C 180,E1 -14604.85,E2 -14604.85} C_VEL
LIN {X 0,Y 343.919,Z 457.556,A -85,B 0,C 180,E1 -14605.795,E2 -14605.795} C_VEL
LIN {X 0,Y 344.766,Z 442.28,A -85,B 0,C 180,E1 -14606.468,E2 -14606.468} C_VEL
LIN {X 0,Y 345.95,Z 413.432,A -85,B 0,C 180,E1 -14607.321,E2 -14607.321} C_VEL
LIN {X 0,Y 350.023,Z 319.09,A -85,B 0,C 180,E1 -14609.936,E2 -14609.936} C_VEL
LIN {X 0,Y 333.736,Z 282.045,A -85,B 0,C 180,E1 -14612.294,E2 -14612.294} C_VEL
LIN {X 0,Y 333.645,Z 281.55,A -85,B 0,C 180,E1 -14612.346,E2 -14612.346} C_VEL
LIN {X 0,Y 333.676,Z 281.546,A -85,B 0,C 180,E1 -14616.137,E2 -14616.137} C_VEL
LIN {X 0,Y 333.633,Z 281.549,A -85,B 0,C 180,E1 -14619.193,E2 -14619.193} C_VEL
LIN {X 0,Y 333.63,Z 281.549,A -85,B 0,C 180,E1 -14622.498,E2 -14622.498} C_VEL
LIN {X 0,Y 333.596,Z 281.557,A -85,B 0,C 180,E1 -14625.953,E2 -14625.953} C_VEL
LIN {X 0,Y 333.646,Z 281.548,A -85,B 0,C 180,E1 -14629.314,E2 -14629.314} C_VEL
LIN {X 0,Y 333.663,Z 281.545,A -85,B 0,C 180,E1 -14633.166,E2 -14633.166} C_VEL
LIN {X 0,Y 333.671,Z 281.545,A -85,B 0,C 180,E1 -14635.339,E2 -14635.339} C_VEL
LIN {X 0,Y 333.626,Z 281.55,A -85,B 0,C 180,E1 -14638.22,E2 -14638.22} C_VEL
LIN {X 0,Y 333.65,Z 281.546,A -85,B 0,C 180,E1 -14641.021,E2 -14641.021} C_VEL
LIN {X 0,Y 333.695,Z 281.541,A -85,B 0,C 180,E1 -14645.087,E2 -14645.087} C_VEL
LIN {X 0,Y 333.665,Z 281.544,A -85,B 0,C 180,E1 -14649.017,E2 -14649.017} C_VEL
LIN {X 0,Y 333.736,Z 281.54,A -85,B 0,C 180,E1 -14651.585,E2 -14651.585} C_VEL
LIN {X 0,Y 333.802,Z 281.532,A -85,B 0,C 180,E1 -14655.575,E2 -14655.575} C_VEL
LIN {X 0,Y 333.827,Z 281.525,A -85,B 0,C 180,E1 -14659.076,E2 -14659.076} C_VEL
LIN {X 0,Y 334.018,Z 281.5,A -85,B 0,C 180,E1 -14662.746,E2 -14662.746} C_VEL
LIN {X 0,Y 333.8,Z 281.529,A -85,B 0,C 180,E1 -14665.167,E2 -14665.167} C_VEL
LIN {X 0,Y 334.096,Z 281.496,A -85,B 0,C 180,E1 -14667.587,E2 -14667.587} C_VEL
LIN {X 0,Y 334.239,Z 281.474,A -85,B 0,C 180,E1 -14669.998,E2 -14669.998} C_VEL
LIN {X 0,Y 334.097,Z 281.49,A -85,B 0,C 180,E1 -14672.41,E2 -14672.41} C_VEL
LIN {X 0,Y 334.015,Z 281.504,A -85,B 0,C 180,E1 -14677.251,E2 -14677.251} C_VEL
LIN {X 0,Y 333.824,Z 281.525,A -85,B 0,C 180,E1 -14680.92,E2 -14680.92} C_VEL
LIN {X 0,Y 333.798,Z 281.527,A -85,B 0,C 180,E1 -14684.633,E2 -14684.633} C_VEL
LIN {X 0,Y 333.785,Z 281.529,A -85,B 0,C 180,E1 -14688.653,E2 -14688.653} C_VEL
LIN {X 0,Y 333.681,Z 281.542,A -85,B 0,C 180,E1 -14692.277,E2 -14692.277} C_VEL
LIN {X 0,Y 333.723,Z 281.537,A -85,B 0,C 180,E1 -14696.245,E2 -14696.245} C_VEL
LIN {X 0,Y 333.677,Z 281.544,A -85,B 0,C 180,E1 -14698.973,E2 -14698.973} C_VEL
LIN {X 0,Y 333.63,Z 281.548,A -85,B 0,C 180,E1 -14702.586,E2 -14702.586} C_VEL
LIN {X 0,Y 333.664,Z 281.544,A -85,B 0,C 180,E1 -14706.138,E2 -14706.138} C_VEL
LIN {X 0,Y 333.634,Z 281.552,A -85,B 0,C 180,E1 -14709.192,E2 -14709.192} C_VEL
LIN {X 0,Y 333.619,Z 281.55,A -85,B 0,C 180,E1 -14712.499,E2 -14712.499} C_VEL
LIN {X 0,Y 333.589,Z 281.552,A -85,B 0,C 180,E1 -14716.301,E2 -14716.301} C_VEL
LIN {X 0,Y 332.916,Z 281.643,A -85,B 0,C 180,E1 -14717.31,E2 -14717.31} C_VEL
LIN {X 0,Y 330.104,Z 281.992,A -85,B 0,C 180,E1 -14718.952,E2 -14718.952} C_VEL
LIN {X 0,Y 327.721,Z 282.291,A -85,B 0,C 180,E1 -14720.281,E2 -14720.281} C_VEL
LIN {X 0,Y 326.687,Z 282.419,A -85,B 0,C 180,E1 -14721.31,E2 -14721.31} C_VEL
LIN {X 0,Y 326.595,Z 282.427,A -85,B 0,C 180,E1 -14721.658,E2 -14721.658} C_VEL
LIN {X 0,Y 326.605,Z 282.426,A -85,B 0,C 180,E1 -14724.851,E2 -14724.851} C_VEL
LIN {X 0,Y 326.593,Z 282.428,A -85,B 0,C 180,E1 -14727.455,E2 -14727.455} C_VEL
LIN {X 0,Y 326.646,Z 282.418,A -85,B 0,C 180,E1 -14730.341,E2 -14730.341} C_VEL
LIN {X 0,Y 326.676,Z 282.415,A -85,B 0,C 180,E1 -14734.516,E2 -14734.516} C_VEL
LIN {X 0,Y 326.605,Z 282.424,A -85,B 0,C 180,E1 -14738.544,E2 -14738.544} C_VEL
LIN {X 0,Y 326.731,Z 282.413,A -85,B 0,C 180,E1 -14741.178,E2 -14741.178} C_VEL
LIN {X 0,Y 326.75,Z 282.408,A -85,B 0,C 180,E1 -14745.434,E2 -14745.434} C_VEL
LIN {X 0,Y 326.756,Z 282.408,A -85,B 0,C 180,E1 -14748.84,E2 -14748.84} C_VEL
LIN {X 0,Y 326.952,Z 282.382,A -85,B 0,C 180,E1 -14752.591,E2 -14752.591} C_VEL
LIN {X 0,Y 326.762,Z 282.41,A -85,B 0,C 180,E1 -14755.066,E2 -14755.066} C_VEL
LIN {X 0,Y 327.034,Z 282.371,A -85,B 0,C 180,E1 -14757.538,E2 -14757.538} C_VEL
LIN {X 0,Y 327.186,Z 282.351,A -85,B 0,C 180,E1 -14760.001,E2 -14760.001} C_VEL
LIN {X 0,Y 327.033,Z 282.371,A -85,B 0,C 180,E1 -14762.464,E2 -14762.464} C_VEL
LIN {X 0,Y 326.983,Z 282.376,A -85,B 0,C 180,E1 -14766.17,E2 -14766.17} C_VEL
LIN {X 0,Y 326.903,Z 282.389,A -85,B 0,C 180,E1 -14768.656,E2 -14768.656} C_VEL
LIN {X 0,Y 326.723,Z 282.41,A -85,B 0,C 180,E1 -14772.423,E2 -14772.423} C_VEL
LIN {X 0,Y 326.743,Z 282.412,A -85,B 0,C 180,E1 -14774.959,E2 -14774.959} C_VEL
LIN {X 0,Y 326.722,Z 282.414,A -85,B 0,C 180,E1 -14778.839,E2 -14778.839} C_VEL
LIN {X 0,Y 326.593,Z 282.43,A -85,B 0,C 180,E1 -14782.79,E2 -14782.79} C_VEL
LIN {X 0,Y 326.68,Z 282.415,A -85,B 0,C 180,E1 -14785.485,E2 -14785.485} C_VEL
LIN {X 0,Y 326.651,Z 282.418,A -85,B 0,C 180,E1 -14789.661,E2 -14789.661} C_VEL
LIN {X 0,Y 326.599,Z 282.424,A -85,B 0,C 180,E1 -14794.021,E2 -14794.021} C_VEL
LIN {X 0,Y 326.619,Z 282.423,A -85,B 0,C 180,E1 -14797.24,E2 -14797.24} C_VEL
LIN {X 0,Y 326.57,Z 282.43,A -85,B 0,C 180,E1 -14801.133,E2 -14801.133} C_VEL
LIN {X 0,Y 326.55,Z 282.436,A -85,B 0,C 180,E1 -14804.75,E2 -14804.75} C_VEL
LIN {X 0,Y 326.57,Z 282.429,A -85,B 0,C 180,E1 -14808.156,E2 -14808.156} C_VEL
LIN {X 0,Y 326.659,Z 282.552,A -85,B 0,C 180,E1 -14810.678,E2 -14810.678} C_VEL
LIN {X 0,Y 330.594,Z 298.372,A -85,B 0,C 180,E1 -14814.396,E2 -14814.396} C_VEL
LIN {X 0,Y 333.743,Z 311.478,A -85,B 0,C 180,E1 -14817.316,E2 -14817.316} C_VEL
LIN {X 0,Y 337.663,Z 322.108,A -85,B 0,C 180,E1 -14817.959,E2 -14817.959} C_VEL
LIN {X 0,Y 343.166,Z 361.318,A -85,B 0,C 180,E1 -14819.605,E2 -14819.605} C_VEL
LIN {X 0,Y 337.819,Z 478.912,A -85,B 0,C 180,E1 -14823.015,E2 -14823.015} C_VEL
LIN {X 0,Y 336.721,Z 494.875,A -85,B 0,C 180,E1 -14823.707,E2 -14823.707} C_VEL
LIN {X 0,Y 335.283,Z 511.04,A -85,B 0,C 180,E1 -14824.668,E2 -14824.668} C_VEL
LIN {X 0,Y 333.864,Z 525.363,A -85,B 0,C 180,E1 -14825.767,E2 -14825.767} C_VEL
LIN {X 0,Y 332.274,Z 539.661,A -85,B 0,C 180,E1 -14827.131,E2 -14827.131} C_VEL
LIN {X 0,Y 330.724,Z 552.792,A -85,B 0,C 180,E1 -14828.661,E2 -14828.661} C_VEL
LIN {X 0,Y 329.273,Z 564.903,A -85,B 0,C 180,E1 -14830.358,E2 -14830.358} C_VEL
LIN {X 0,Y 328.019,Z 576.037,A -85,B 0,C 180,E1 -14832.225,E2 -14832.225} C_VEL
LIN {X 0,Y 326.975,Z 585.437,A -85,B 0,C 180,E1 -14834.097,E2 -14834.097} C_VEL
LIN {X 0,Y 326.1,Z 594.633,A -85,B 0,C 180,E1 -14836.288,E2 -14836.288} C_VEL
LIN {X 0,Y 325.664,Z 601.267,A -85,B 0,C 180,E1 -14838.171,E2 -14838.171} C_VEL
LIN {X 0,Y 325.237,Z 608.388,A -85,B 0,C 180,E1 -14840.675,E2 -14840.675} C_VEL
LIN {X 0,Y 325.156,Z 613.873,A -85,B 0,C 180,E1 -14843.174,E2 -14843.174} C_VEL
LIN {X 0,Y 325.134,Z 616.961,A -85,B 0,C 180,E1 -14845.042,E2 -14845.042} C_VEL
LIN {X 0,Y 325.143,Z 619.839,A -85,B 0,C 180,E1 -14847.524,E2 -14847.524} C_VEL
LIN {X 0,Y 325.235,Z 620.764,A -85,B 0,C 180,E1 -14848.764,E2 -14848.764} C_VEL
LIN {X 0,Y 325.193,Z 621.588,A -85,B 0,C 180,E1 -14851.24,E2 -14851.24} C_VEL
LIN {X 0,Y 324.987,Z 621.085,A -85,B 0,C 180,E1 -14853.721,E2 -14853.721} C_VEL
LIN {X 0,Y 324.966,Z 619.293,A -85,B 0,C 180,E1 -14856.209,E2 -14856.209} C_VEL
LIN {X 0,Y 325.103,Z 616.183,A -85,B 0,C 180,E1 -14858.705,E2 -14858.705} C_VEL
LIN {X 0,Y 325.504,Z 611.74,A -85,B 0,C 180,E1 -14861.207,E2 -14861.207} C_VEL
LIN {X 0,Y 326.35,Z 605.913,A -85,B 0,C 180,E1 -14863.704,E2 -14863.704} C_VEL
LIN {X 0,Y 327.704,Z 598.585,A -85,B 0,C 180,E1 -14866.19,E2 -14866.19} C_VEL
LIN {X 0,Y 329.563,Z 589.602,A -85,B 0,C 180,E1 -14868.657,E2 -14868.657} C_VEL
LIN {X 0,Y 331.605,Z 580.178,A -85,B 0,C 180,E1 -14870.795,E2 -14870.795} C_VEL
LIN {X 0,Y 334.268,Z 569.036,A -85,B 0,C 180,E1 -14872.891,E2 -14872.891} C_VEL
LIN {X 0,Y 337.329,Z 555.852,A -85,B 0,C 180,E1 -14874.956,E2 -14874.956} C_VEL
LIN {X 0,Y 340.492,Z 542.377,A -85,B 0,C 180,E1 -14876.677,E2 -14876.677} C_VEL
LIN {X 0,Y 343.782,Z 527.573,A -85,B 0,C 180,E1 -14878.231,E2 -14878.231} C_VEL
LIN {X 0,Y 347.362,Z 510.6,A -85,B 0,C 180,E1 -14879.65,E2 -14879.65} C_VEL
LIN {X 0,Y 350.201,Z 495.937,A -85,B 0,C 180,E1 -14880.615,E2 -14880.615} C_VEL
LIN {X 0,Y 353.123,Z 478.637,A -85,B 0,C 180,E1 -14881.497,E2 -14881.497} C_VEL
LIN {X 0,Y 355.609,Z 458.139,A -85,B 0,C 180,E1 -14882.293,E2 -14882.293} C_VEL
LIN {X 0,Y 363.743,Z 392.068,A -85,B 0,C 180,E1 -14884.637,E2 -14884.637} C_VEL
LIN {X 0,Y 367.251,Z 366.098,A -85,B 0,C 180,E1 -14885.594,E2 -14885.594} C_VEL
LIN {X 0,Y 367.26,Z 353.249,A -85,B 0,C 180,E1 -14886.602,E2 -14886.602} C_VEL
LIN {X 0,Y 367.114,Z 350.918,A -85,B 0,C 180,E1 -14886.842,E2 -14886.842} C_VEL
LIN {X 0,Y 365.408,Z 345.69,A -85,B 0,C 180,E1 -14887.894,E2 -14887.894} C_VEL
LIN {X 0,Y 364.107,Z 342.032,A -85,B 0,C 180,E1 -14888.77,E2 -14888.77} C_VEL
LIN {X 0,Y 362.081,Z 336.658,A -85,B 0,C 180,E1 -14890.408,E2 -14890.408} C_VEL
LIN {X 0,Y 360.221,Z 331.826,A -85,B 0,C 180,E1 -14892.615,E2 -14892.615} C_VEL
LIN {X 0,Y 359.589,Z 329.452,A -85,B 0,C 180,E1 -14894.296,E2 -14894.296} C_VEL
LIN {X 0,Y 359.486,Z 328.729,A -85,B 0,C 180,E1 -14895.266,E2 -14895.266} C_VEL
LIN {X 0,Y 359.933,Z 328.789,A -85,B 0,C 180,E1 -14897.393,E2 -14897.393} C_VEL
LIN {X 0,Y 361.884,Z 330.351,A -85,B 0,C 180,E1 -14899.767,E2 -14899.767} C_VEL
LIN {X 0,Y 364.224,Z 333.675,A -85,B 0,C 180,E1 -14901.614,E2 -14901.614} C_VEL
LIN {X 0,Y 366.446,Z 337.234,A -85,B 0,C 180,E1 -14902.967,E2 -14902.967} C_VEL
LIN {X 0,Y 369.071,Z 341.979,A -85,B 0,C 180,E1 -14904.319,E2 -14904.319} C_VEL
LIN {X 0,Y 369.682,Z 343.406,A -85,B 0,C 180,E1 -14904.627,E2 -14904.627} C_VEL
LIN {X 0,Y 359.722,Z 414.596,A -85,B 0,C 180,E1 -14907.21,E2 -14907.21} C_VEL
LIN {X 0,Y 355.334,Z 450.98,A -85,B 0,C 180,E1 -14908.554,E2 -14908.554} C_VEL
LIN {X 0,Y 353.123,Z 467.019,A -85,B 0,C 180,E1 -14909.385,E2 -14909.385} C_VEL
LIN {X 0,Y 350.602,Z 482.352,A -85,B 0,C 180,E1 -14910.42,E2 -14910.42} C_VEL
LIN {X 0,Y 347.895,Z 496.875,A -85,B 0,C 180,E1 -14911.657,E2 -14911.657} C_VEL
LIN {X 0,Y 344.825,Z 511.547,A -85,B 0,C 180,E1 -14913.195,E2 -14913.195} C_VEL
LIN {X 0,Y 341.72,Z 524.932,A -85,B 0,C 180,E1 -14914.928,E2 -14914.928} C_VEL
LIN {X 0,Y 338.677,Z 536.8,A -85,B 0,C 180,E1 -14916.778,E2 -14916.778} C_VEL
LIN {X 0,Y 335.905,Z 547.608,A -85,B 0,C 180,E1 -14918.843,E2 -14918.843} C_VEL
LIN {X 0,Y 333.494,Z 556.653,A -85,B 0,C 180,E1 -14920.934,E2 -14920.934} C_VEL
LIN {X 0,Y 331.035,Z 565.215,A -85,B 0,C 180,E1 -14923.344,E2 -14923.344} C_VEL
LIN {X 0,Y 329.212,Z 572.065,A -85,B 0,C 180,E1 -14925.788,E2 -14925.788} C_VEL
LIN {X 0,Y 327.739,Z 577.429,A -85,B 0,C 180,E1 -14928.245,E2 -14928.245} C_VEL
LIN {X 0,Y 327.012,Z 580.566,A -85,B 0,C 180,E1 -14930.099,E2 -14930.099} C_VEL
LIN {X 0,Y 326.121,Z 583.592,A -85,B 0,C 180,E1 -14932.57,E2 -14932.57} C_VEL
LIN {X 0,Y 325.543,Z 585.344,A -85,B 0,C 180,E1 -14935.045,E2 -14935.045} C_VEL
LIN {X 0,Y 325.407,Z 585.857,A -85,B 0,C 180,E1 -14937.523,E2 -14937.523} C_VEL
LIN {X 0,Y 325.149,Z 585.151,A -85,B 0,C 180,E1 -14939.999,E2 -14939.999} C_VEL
LIN {X 0,Y 325.134,Z 583.194,A -85,B 0,C 180,E1 -14942.477,E2 -14942.477} C_VEL
LIN {X 0,Y 325.244,Z 579.941,A -85,B 0,C 180,E1 -14944.957,E2 -14944.957} C_VEL
LIN {X 0,Y 325.476,Z 575.317,A -85,B 0,C 180,E1 -14947.443,E2 -14947.443} C_VEL
LIN {X 0,Y 325.868,Z 569.196,A -85,B 0,C 180,E1 -14949.934,E2 -14949.934} C_VEL
LIN {X 0,Y 326.638,Z 561.414,A -85,B 0,C 180,E1 -14952.424,E2 -14952.424} C_VEL
LIN {X 0,Y 327.511,Z 553.037,A -85,B 0,C 180,E1 -14954.603,E2 -14954.603} C_VEL
LIN {X 0,Y 328.573,Z 542.926,A -85,B 0,C 180,E1 -14956.782,E2 -14956.782} C_VEL
LIN {X 0,Y 329.748,Z 532.59,A -85,B 0,C 180,E1 -14958.643,E2 -14958.643} C_VEL
LIN {X 0,Y 331.199,Z 520.312,A -85,B 0,C 180,E1 -14960.494,E2 -14960.494} C_VEL
LIN {X 0,Y 332.678,Z 506.93,A -85,B 0,C 180,E1 -14962.169,E2 -14962.169} C_VEL
LIN {X 0,Y 334.122,Z 493.486,A -85,B 0,C 180,E1 -14963.555,E2 -14963.555} C_VEL
LIN {X 0,Y 335.482,Z 479.061,A -85,B 0,C 180,E1 -14964.769,E2 -14964.769} C_VEL
LIN {X 0,Y 336.768,Z 463.177,A -85,B 0,C 180,E1 -14965.825,E2 -14965.825} C_VEL
LIN {X 0,Y 337.691,Z 447.043,A -85,B 0,C 180,E1 -14966.631,E2 -14966.631} C_VEL
LIN {X 0,Y 338.519,Z 429.828,A -85,B 0,C 180,E1 -14967.218,E2 -14967.218} C_VEL
LIN {X 0,Y 343.431,Z 321.001,A -85,B 0,C 180,E1 -14970.324,E2 -14970.324} C_VEL
LIN {X 0,Y 326.669,Z 282.835,A -85,B 0,C 180,E1 -14972.815,E2 -14972.815} C_VEL
LIN {X 0,Y 326.601,Z 282.427,A -85,B 0,C 180,E1 -14972.895,E2 -14972.895} C_VEL
LIN {X 0,Y 326.613,Z 282.425,A -85,B 0,C 180,E1 -14975.518,E2 -14975.518} C_VEL
LIN {X 0,Y 326.599,Z 282.425,A -85,B 0,C 180,E1 -14979.223,E2 -14979.223} C_VEL
LIN {X 0,Y 326.574,Z 282.427,A -85,B 0,C 180,E1 -14982.97,E2 -14982.97} C_VEL
LIN {X 0,Y 326.575,Z 282.427,A -85,B 0,C 180,E1 -14987.026,E2 -14987.026} C_VEL
LIN {X 0,Y 326.61,Z 282.423,A -85,B 0,C 180,E1 -14990.771,E2 -14990.771} C_VEL
LIN {X 0,Y 326.61,Z 282.423,A -85,B 0,C 180,E1 -14994.478,E2 -14994.478} C_VEL
LIN {X 0,Y 326.605,Z 282.426,A -85,B 0,C 180,E1 -14997.454,E2 -14997.454} C_VEL
LIN {X 0,Y 326.613,Z 282.423,A -85,B 0,C 180,E1 -15000.335,E2 -15000.335} C_VEL
LIN {X 0,Y 326.639,Z 282.419,A -85,B 0,C 180,E1 -15004.642,E2 -15004.642} C_VEL
LIN {X 0,Y 326.613,Z 282.422,A -85,B 0,C 180,E1 -15008.541,E2 -15008.541} C_VEL
LIN {X 0,Y 326.658,Z 282.417,A -85,B 0,C 180,E1 -15012.468,E2 -15012.468} C_VEL
LIN {X 0,Y 326.753,Z 282.405,A -85,B 0,C 180,E1 -15016.313,E2 -15016.313} C_VEL
LIN {X 0,Y 326.807,Z 282.4,A -85,B 0,C 180,E1 -15020.092,E2 -15020.092} C_VEL
LIN {X 0,Y 326.972,Z 282.378,A -85,B 0,C 180,E1 -15022.589,E2 -15022.589} C_VEL
LIN {X 0,Y 326.767,Z 282.405,A -85,B 0,C 180,E1 -15025.063,E2 -15025.063} C_VEL
LIN {X 0,Y 327.037,Z 282.375,A -85,B 0,C 180,E1 -15027.535,E2 -15027.535} C_VEL
LIN {X 0,Y 327.19,Z 282.352,A -85,B 0,C 180,E1 -15029.998,E2 -15029.998} C_VEL
LIN {X 0,Y 327.037,Z 282.37,A -85,B 0,C 180,E1 -15032.462,E2 -15032.462} C_VEL
LIN {X 0,Y 326.986,Z 282.377,A -85,B 0,C 180,E1 -15036.168,E2 -15036.168} C_VEL
LIN {X 0,Y 326.905,Z 282.386,A -85,B 0,C 180,E1 -15038.654,E2 -15038.654} C_VEL
LIN {X 0,Y 326.724,Z 282.409,A -85,B 0,C 180,E1 -15042.42,E2 -15042.42} C_VEL
LIN {X 0,Y 326.744,Z 282.408,A -85,B 0,C 180,E1 -15044.956,E2 -15044.956} C_VEL
LIN {X 0,Y 326.722,Z 282.41,A -85,B 0,C 180,E1 -15048.837,E2 -15048.837} C_VEL
LIN {X 0,Y 326.61,Z 282.424,A -85,B 0,C 180,E1 -15052.786,E2 -15052.786} C_VEL
LIN {X 0,Y 326.678,Z 282.419,A -85,B 0,C 180,E1 -15055.483,E2 -15055.483} C_VEL
LIN {X 0,Y 326.635,Z 282.423,A -85,B 0,C 180,E1 -15059.659,E2 -15059.659} C_VEL
LIN {X 0,Y 326.594,Z 282.425,A -85,B 0,C 180,E1 -15064.018,E2 -15064.018} C_VEL
LIN {X 0,Y 326.616,Z 282.427,A -85,B 0,C 180,E1 -15067.238,E2 -15067.238} C_VEL
LIN {X 0,Y 326.565,Z 282.432,A -85,B 0,C 180,E1 -15071.131,E2 -15071.131} C_VEL
LIN {X 0,Y 326.543,Z 282.432,A -85,B 0,C 180,E1 -15074.747,E2 -15074.747} C_VEL
LIN {X 0,Y 326.562,Z 282.429,A -85,B 0,C 180,E1 -15078.154,E2 -15078.154} C_VEL
LIN {X 0,Y 326.595,Z 282.427,A -85,B 0,C 180,E1 -15081.658,E2 -15081.658} C_VEL
LIN {X 0,Y 325.916,Z 282.512,A -85,B 0,C 180,E1 -15082.688,E2 -15082.688} C_VEL
LIN {X 0,Y 323.086,Z 282.862,A -85,B 0,C 180,E1 -15084.364,E2 -15084.364} C_VEL
LIN {X 0,Y 320.681,Z 283.163,A -85,B 0,C 180,E1 -15085.722,E2 -15085.722} C_VEL
LIN {X 0,Y 319.627,Z 283.295,A -85,B 0,C 180,E1 -15086.772,E2 -15086.772} C_VEL
LIN {X 0,Y 319.527,Z 283.303,A -85,B 0,C 180,E1 -15087.128,E2 -15087.128} C_VEL
LIN {X 0,Y 319.575,Z 283.304,A -85,B 0,C 180,E1 -15091.066,E2 -15091.066} C_VEL
LIN {X 0,Y 319.62,Z 283.294,A -85,B 0,C 180,E1 -15094.355,E2 -15094.355} C_VEL
LIN {X 0,Y 319.554,Z 283.302,A -85,B 0,C 180,E1 -15098.046,E2 -15098.046} C_VEL
LIN {X 0,Y 319.675,Z 283.291,A -85,B 0,C 180,E1 -15100.963,E2 -15100.963} C_VEL
LIN {X 0,Y 319.717,Z 283.285,A -85,B 0,C 180,E1 -15105.276,E2 -15105.276} C_VEL
LIN {X 0,Y 319.743,Z 283.278,A -85,B 0,C 180,E1 -15109.874,E2 -15109.874} C_VEL
LIN {X 0,Y 319.912,Z 283.258,A -85,B 0,C 180,E1 -15112.427,E2 -15112.427} C_VEL
LIN {X 0,Y 319.732,Z 283.285,A -85,B 0,C 180,E1 -15114.957,E2 -15114.957} C_VEL
LIN {X 0,Y 319.978,Z 283.251,A -85,B 0,C 180,E1 -15117.483,E2 -15117.483} C_VEL
LIN {X 0,Y 320.138,Z 283.229,A -85,B 0,C 180,E1 -15120.001,E2 -15120.001} C_VEL
LIN {X 0,Y 319.976,Z 283.251,A -85,B 0,C 180,E1 -15122.519,E2 -15122.519} C_VEL
LIN {X 0,Y 319.939,Z 283.254,A -85,B 0,C 180,E1 -15126.307,E2 -15126.307} C_VEL
LIN {X 0,Y 319.832,Z 283.272,A -85,B 0,C 180,E1 -15128.849,E2 -15128.849} C_VEL
LIN {X 0,Y 319.671,Z 283.291,A -85,B 0,C 180,E1 -15132.701,E2 -15132.701} C_VEL
LIN {X 0,Y 319.689,Z 283.287,A -85,B 0,C 180,E1 -15135.297,E2 -15135.297} C_VEL
LIN {X 0,Y 319.641,Z 283.293,A -85,B 0,C 180,E1 -15139.258,E2 -15139.258} C_VEL
LIN {X 0,Y 319.55,Z 283.304,A -85,B 0,C 180,E1 -15143.322,E2 -15143.322} C_VEL
LIN {X 0,Y 319.609,Z 283.295,A -85,B 0,C 180,E1 -15146.091,E2 -15146.091} C_VEL
LIN {X 0,Y 319.581,Z 283.303,A -85,B 0,C 180,E1 -15148.935,E2 -15148.935} C_VEL
LIN {X 0,Y 319.524,Z 283.306,A -85,B 0,C 180,E1 -15151.864,E2 -15151.864} C_VEL
LIN {X 0,Y 319.571,Z 283.3,A -85,B 0,C 180,E1 -15155.545,E2 -15155.545} C_VEL
LIN {X 0,Y 319.551,Z 283.302,A -85,B 0,C 180,E1 -15159.671,E2 -15159.671} C_VEL
LIN {X 0,Y 319.551,Z 283.302,A -85,B 0,C 180,E1 -15163.469,E2 -15163.469} C_VEL
LIN {X 0,Y 319.554,Z 283.305,A -85,B 0,C 180,E1 -15167.019,E2 -15167.019} C_VEL
LIN {X 0,Y 319.587,Z 283.434,A -85,B 0,C 180,E1 -15170.234,E2 -15170.234} C_VEL
LIN {X 0,Y 323.33,Z 298.375,A -85,B 0,C 180,E1 -15173.831,E2 -15173.831} C_VEL
LIN {X 0,Y 326.374,Z 311.018,A -85,B 0,C 180,E1 -15176.718,E2 -15176.718} C_VEL
LIN {X 0,Y 331.287,Z 324.384,A -85,B 0,C 180,E1 -15177.57,E2 -15177.57} C_VEL
LIN {X 0,Y 336.521,Z 361.161,A -85,B 0,C 180,E1 -15179.162,E2 -15179.162} C_VEL
LIN {X 0,Y 331.03,Z 478.625,A -85,B 0,C 180,E1 -15182.672,E2 -15182.672} C_VEL
LIN {X 0,Y 329.96,Z 493.933,A -85,B 0,C 180,E1 -15183.347,E2 -15183.347} C_VEL
LIN {X 0,Y 328.525,Z 509.214,A -85,B 0,C 180,E1 -15184.257,E2 -15184.257} C_VEL
LIN {X 0,Y 327.075,Z 524.018,A -85,B 0,C 180,E1 -15185.4,E2 -15185.4} C_VEL
LIN {X 0,Y 325.429,Z 538.46,A -85,B 0,C 180,E1 -15186.79,E2 -15186.79} C_VEL
LIN {X 0,Y 323.832,Z 551.714,A -85,B 0,C 180,E1 -15188.352,E2 -15188.352} C_VEL
LIN {X 0,Y 322.223,Z 564.944,A -85,B 0,C 180,E1 -15190.243,E2 -15190.243} C_VEL
LIN {X 0,Y 320.926,Z 576.004,A -85,B 0,C 180,E1 -15192.148,E2 -15192.148} C_VEL
LIN {X 0,Y 319.878,Z 585.348,A -85,B 0,C 180,E1 -15194.062,E2 -15194.062} C_VEL
LIN {X 0,Y 319.023,Z 594.497,A -85,B 0,C 180,E1 -15196.303,E2 -15196.303} C_VEL
LIN {X 0,Y 318.471,Z 602.03,A -85,B 0,C 180,E1 -15198.546,E2 -15198.546} C_VEL
LIN {X 0,Y 318.134,Z 608.908,A -85,B 0,C 180,E1 -15201.106,E2 -15201.106} C_VEL
LIN {X 0,Y 318.085,Z 614.148,A -85,B 0,C 180,E1 -15203.659,E2 -15203.659} C_VEL
LIN {X 0,Y 318.077,Z 616.189,A -85,B 0,C 180,E1 -15204.931,E2 -15204.931} C_VEL
LIN {X 0,Y 318.056,Z 619.185,A -85,B 0,C 180,E1 -15207.469,E2 -15207.469} C_VEL
LIN {X 0,Y 318.176,Z 620.172,A -85,B 0,C 180,E1 -15208.736,E2 -15208.736} C_VEL
LIN {X 0,Y 318.113,Z 621.111,A -85,B 0,C 180,E1 -15211.268,E2 -15211.268} C_VEL
LIN {X 0,Y 317.911,Z 620.718,A -85,B 0,C 180,E1 -15213.804,E2 -15213.804} C_VEL
LIN {X 0,Y 317.882,Z 619.002,A -85,B 0,C 180,E1 -15216.348,E2 -15216.348} C_VEL
LIN {X 0,Y 318.038,Z 615.992,A -85,B 0,C 180,E1 -15218.9,E2 -15218.9} C_VEL
LIN {X 0,Y 318.492,Z 611.686,A -85,B 0,C 180,E1 -15221.457,E2 -15221.457} C_VEL
LIN {X 0,Y 319.405,Z 606.011,A -85,B 0,C 180,E1 -15224.008,E2 -15224.008} C_VEL
LIN {X 0,Y 320.862,Z 598.856,A -85,B 0,C 180,E1 -15226.545,E2 -15226.545} C_VEL
LIN {X 0,Y 322.84,Z 590.077,A -85,B 0,C 180,E1 -15229.06,E2 -15229.06} C_VEL
LIN {X 0,Y 325.003,Z 580.896,A -85,B 0,C 180,E1 -15231.237,E2 -15231.237} C_VEL
LIN {X 0,Y 327.815,Z 570.047,A -85,B 0,C 180,E1 -15233.369,E2 -15233.369} C_VEL
LIN {X 0,Y 331.045,Z 557.232,A -85,B 0,C 180,E1 -15235.463,E2 -15235.463} C_VEL
LIN {X 0,Y 334.331,Z 544.259,A -85,B 0,C 180,E1 -15237.209,E2 -15237.209} C_VEL
LIN {X 0,Y 337.828,Z 529.904,A -85,B 0,C 180,E1 -15238.802,E2 -15238.802} C_VEL
LIN {X 0,Y 341.244,Z 515.28,A -85,B 0,C 180,E1 -15240.116,E2 -15240.116} C_VEL
LIN {X 0,Y 344.576,Z 499.508,A -85,B 0,C 180,E1 -15241.255,E2 -15241.255} C_VEL
LIN {X 0,Y 348.01,Z 481.003,A -85,B 0,C 180,E1 -15242.271,E2 -15242.271} C_VEL
LIN {X 0,Y 350.683,Z 462.194,A -85,B 0,C 180,E1 -15243.059,E2 -15243.059} C_VEL
LIN {X 0,Y 358.925,Z 399.595,A -85,B 0,C 180,E1 -15245.328,E2 -15245.328} C_VEL
LIN {X 0,Y 363.569,Z 367.912,A -85,B 0,C 180,E1 -15246.505,E2 -15246.505} C_VEL
LIN {X 0,Y 363.808,Z 355.66,A -85,B 0,C 180,E1 -15247.504,E2 -15247.504} C_VEL
LIN {X 0,Y 362.287,Z 350.44,A -85,B 0,C 180,E1 -15248.602,E2 -15248.602} C_VEL
LIN {X 0,Y 361.045,Z 346.79,A -85,B 0,C 180,E1 -15249.574,E2 -15249.574} C_VEL
LIN {X 0,Y 359.755,Z 342.907,A -85,B 0,C 180,E1 -15250.804,E2 -15250.804} C_VEL
LIN {X 0,Y 358.202,Z 338.251,A -85,B 0,C 180,E1 -15252.988,E2 -15252.988} C_VEL
LIN {X 0,Y 357.752,Z 336.094,A -85,B 0,C 180,E1 -15254.597,E2 -15254.597} C_VEL
LIN {X 0,Y 357.728,Z 335.492,A -85,B 0,C 180,E1 -15255.945,E2 -15255.945} C_VEL
LIN {X 0,Y 358.405,Z 335.914,A -85,B 0,C 180,E1 -15257.854,E2 -15257.854} C_VEL
LIN {X 0,Y 359.969,Z 337.266,A -85,B 0,C 180,E1 -15259.684,E2 -15259.684} C_VEL
LIN {X 0,Y 362.013,Z 340.275,A -85,B 0,C 180,E1 -15261.389,E2 -15261.389} C_VEL
LIN {X 0,Y 363.812,Z 343.354,A -85,B 0,C 180,E1 -15262.577,E2 -15262.577} C_VEL
LIN {X 0,Y 365.927,Z 347.42,A -85,B 0,C 180,E1 -15263.772,E2 -15263.772} C_VEL
LIN {X 0,Y 354.881,Z 421.095,A -85,B 0,C 180,E1 -15266.493,E2 -15266.493} C_VEL
LIN {X 0,Y 350.844,Z 452.283,A -85,B 0,C 180,E1 -15267.692,E2 -15267.692} C_VEL
LIN {X 0,Y 348.419,Z 468.183,A -85,B 0,C 180,E1 -15268.538,E2 -15268.538} C_VEL
LIN {X 0,Y 345.648,Z 483.687,A -85,B 0,C 180,E1 -15269.616,E2 -15269.616} C_VEL
LIN {X 0,Y 342.763,Z 497.903,A -85,B 0,C 180,E1 -15270.858,E2 -15270.858} C_VEL
LIN {X 0,Y 339.494,Z 512.344,A -85,B 0,C 180,E1 -15272.406,E2 -15272.406} C_VEL
LIN {X 0,Y 336.223,Z 525.465,A -85,B 0,C 180,E1 -15274.138,E2 -15274.138} C_VEL
LIN {X 0,Y 332.92,Z 537.355,A -85,B 0,C 180,E1 -15276.022,E2 -15276.022} C_VEL
LIN {X 0,Y 329.932,Z 548.103,A -85,B 0,C 180,E1 -15278.112,E2 -15278.112} C_VEL
LIN {X 0,Y 327.327,Z 557.113,A -85,B 0,C 180,E1 -15280.234,E2 -15280.234} C_VEL
LIN {X 0,Y 324.958,Z 564.684,A -85,B 0,C 180,E1 -15282.374,E2 -15282.374} C_VEL
LIN {X 0,Y 323.297,Z 570.134,A -85,B 0,C 180,E1 -15284.232,E2 -15284.232} C_VEL
LIN {X 0,Y 321.501,Z 576.045,A -85,B 0,C 180,E1 -15286.73,E2 -15286.73} C_VEL
LIN {X 0,Y 320.609,Z 579.511,A -85,B 0,C 180,E1 -15288.621,E2 -15288.621} C_VEL
LIN {X 0,Y 319.565,Z 583.029,A -85,B 0,C 180,E1 -15291.143,E2 -15291.143} C_VEL
LIN {X 0,Y 318.713,Z 585.307,A -85,B 0,C 180,E1 -15293.669,E2 -15293.669} C_VEL
LIN {X 0,Y 318.429,Z 586.309,A -85,B 0,C 180,E1 -15296.203,E2 -15296.203} C_VEL
LIN {X 0,Y 318.17,Z 586.076,A -85,B 0,C 180,E1 -15298.733,E2 -15298.733} C_VEL
LIN {X 0,Y 318.034,Z 584.609,A -85,B 0,C 180,E1 -15301.265,E2 -15301.265} C_VEL
LIN {X 0,Y 318.091,Z 581.871,A -85,B 0,C 180,E1 -15303.799,E2 -15303.799} C_VEL
LIN {X 0,Y 318.291,Z 577.555,A -85,B 0,C 180,E1 -15306.466,E2 -15306.466} C_VEL
LIN {X 0,Y 318.587,Z 572.284,A -85,B 0,C 180,E1 -15308.882,E2 -15308.882} C_VEL
LIN {X 0,Y 319.115,Z 565.185,A -85,B 0,C 180,E1 -15311.431,E2 -15311.431} C_VEL
LIN {X 0,Y 319.998,Z 557.502,A -85,B 0,C 180,E1 -15313.655,E2 -15313.655} C_VEL
LIN {X 0,Y 320.96,Z 548.214,A -85,B 0,C 180,E1 -15315.883,E2 -15315.883} C_VEL
LIN {X 0,Y 322.093,Z 538.746,A -85,B 0,C 180,E1 -15317.786,E2 -15317.786} C_VEL
LIN {X 0,Y 323.554,Z 526.527,A -85,B 0,C 180,E1 -15319.839,E2 -15319.839} C_VEL
LIN {X 0,Y 324.968,Z 514.14,A -85,B 0,C 180,E1 -15321.57,E2 -15321.57} C_VEL
LIN {X 0,Y 326.527,Z 500.7,A -85,B 0,C 180,E1 -15323.128,E2 -15323.128} C_VEL
LIN {X 0,Y 327.987,Z 485.978,A -85,B 0,C 180,E1 -15324.528,E2 -15324.528} C_VEL
LIN {X 0,Y 329.365,Z 470.725,A -85,B 0,C 180,E1 -15325.684,E2 -15325.684} C_VEL
LIN {X 0,Y 330.479,Z 454.335,A -85,B 0,C 180,E1 -15326.638,E2 -15326.638} C_VEL
LIN {X 0,Y 331.422,Z 437.967,A -85,B 0,C 180,E1 -15327.319,E2 -15327.319} C_VEL
LIN {X 0,Y 336.813,Z 323.423,A -85,B 0,C 180,E1 -15330.699,E2 -15330.699} C_VEL
LIN {X 0,Y 327.417,Z 301.522,A -85,B 0,C 180,E1 -15332.112,E2 -15332.112} C_VEL
LIN {X 0,Y 319.656,Z 283.892,A -85,B 0,C 180,E1 -15333.333,E2 -15333.333} C_VEL
LIN {X 0,Y 319.57,Z 283.303,A -85,B 0,C 180,E1 -15333.399,E2 -15333.399} C_VEL
LIN {X 0,Y 319.557,Z 283.303,A -85,B 0,C 180,E1 -15336.426,E2 -15336.426} C_VEL
LIN {X 0,Y 319.559,Z 283.305,A -85,B 0,C 180,E1 -15339.667,E2 -15339.667} C_VEL
LIN {X 0,Y 319.52,Z 283.308,A -85,B 0,C 180,E1 -15343.459,E2 -15343.459} C_VEL
LIN {X 0,Y 319.553,Z 283.302,A -85,B 0,C 180,E1 -15347.015,E2 -15347.015} C_VEL
LIN {X 0,Y 319.545,Z 283.304,A -85,B 0,C 180,E1 -15350.369,E2 -15350.369} C_VEL
LIN {X 0,Y 319.556,Z 283.305,A -85,B 0,C 180,E1 -15353.57,E2 -15353.57} C_VEL
LIN {X 0,Y 319.575,Z 283.299,A -85,B 0,C 180,E1 -15356.685,E2 -15356.685} C_VEL
LIN {X 0,Y 319.557,Z 283.306,A -85,B 0,C 180,E1 -15359.611,E2 -15359.611} C_VEL
LIN {X 0,Y 319.542,Z 283.303,A -85,B 0,C 180,E1 -15362.49,E2 -15362.49} C_VEL
LIN {X 0,Y 319.571,Z 283.302,A -85,B 0,C 180,E1 -15365.3,E2 -15365.3} C_VEL
LIN {X 0,Y 319.563,Z 283.303,A -85,B 0,C 180,E1 -15368.044,E2 -15368.044} C_VEL
LIN {X 0,Y 319.608,Z 283.297,A -85,B 0,C 180,E1 -15372.069,E2 -15372.069} C_VEL
LIN {X 0,Y 319.726,Z 283.283,A -85,B 0,C 180,E1 -15376.006,E2 -15376.006} C_VEL
LIN {X 0,Y 319.752,Z 283.281,A -85,B 0,C 180,E1 -15379.871,E2 -15379.871} C_VEL
LIN {X 0,Y 319.926,Z 283.256,A -85,B 0,C 180,E1 -15382.424,E2 -15382.424} C_VEL
LIN {X 0,Y 319.737,Z 283.28,A -85,B 0,C 180,E1 -15384.954,E2 -15384.954} C_VEL
LIN {X 0,Y 319.981,Z 283.254,A -85,B 0,C 180,E1 -15387.481,E2 -15387.481} C_VEL
LIN {X 0,Y 320.142,Z 283.23,A -85,B 0,C 180,E1 -15389.998,E2 -15389.998} C_VEL
LIN {X 0,Y 319.981,Z 283.248,A -85,B 0,C 180,E1 -15392.516,E2 -15392.516} C_VEL
LIN {X 0,Y 319.942,Z 283.254,A -85,B 0,C 180,E1 -15396.304,E2 -15396.304} C_VEL
LIN {X 0,Y 319.833,Z 283.268,A -85,B 0,C 180,E1 -15398.846,E2 -15398.846} C_VEL
LIN {X 0,Y 319.671,Z 283.287,A -85,B 0,C 180,E1 -15402.698,E2 -15402.698} C_VEL
LIN {X 0,Y 319.689,Z 283.289,A -85,B 0,C 180,E1 -15405.294,E2 -15405.294} C_VEL
LIN {X 0,Y 319.663,Z 283.292,A -85,B 0,C 180,E1 -15409.254,E2 -15409.254} C_VEL
LIN {X 0,Y 319.559,Z 283.306,A -85,B 0,C 180,E1 -15413.318,E2 -15413.318} C_VEL
LIN {X 0,Y 319.606,Z 283.296,A -85,B 0,C 180,E1 -15416.088,E2 -15416.088} C_VEL
LIN {X 0,Y 319.567,Z 283.302,A -85,B 0,C 180,E1 -15418.933,E2 -15418.933} C_VEL
LIN {X 0,Y 319.518,Z 283.308,A -85,B 0,C 180,E1 -15421.861,E2 -15421.861} C_VEL
LIN {X 0,Y 319.568,Z 283.304,A -85,B 0,C 180,E1 -15425.542,E2 -15425.542} C_VEL
LIN {X 0,Y 319.545,Z 283.303,A -85,B 0,C 180,E1 -15428.009,E2 -15428.009} C_VEL
LIN {X 0,Y 319.512,Z 283.31,A -85,B 0,C 180,E1 -15431.596,E2 -15431.596} C_VEL
LIN {X 0,Y 319.502,Z 283.314,A -85,B 0,C 180,E1 -15435.262,E2 -15435.262} C_VEL
LIN {X 0,Y 319.514,Z 283.308,A -85,B 0,C 180,E1 -15438.711,E2 -15438.711} C_VEL
LIN {X 0,Y 319.547,Z 283.303,A -85,B 0,C 180,E1 -15442.348,E2 -15442.348} C_VEL
LIN {X 0,Y 319.546,Z 283.308,A -85,B 0,C 180,E1 -15445.123,E2 -15445.123} C_VEL
LIN {X 0,Y 319.527,Z 283.303,A -85,B 0,C 180,E1 -15447.128,E2 -15447.128} C_VEL
LIN {X 0,Y 318.828,Z 283.393,A -85,B 0,C 180,E1 -15448.18,E2 -15448.18} C_VEL
LIN {X 0,Y 315.986,Z 283.747,A -85,B 0,C 180,E1 -15449.894,E2 -15449.894} C_VEL
LIN {X 0,Y 313.612,Z 284.047,A -85,B 0,C 180,E1 -15451.284,E2 -15451.284} C_VEL
LIN {X 0,Y 312.614,Z 284.166,A -85,B 0,C 180,E1 -15452.358,E2 -15452.358} C_VEL
LIN {X 0,Y 312.541,Z 284.176,A -85,B 0,C 180,E1 -15452.722,E2 -15452.722} C_VEL
LIN {X 0,Y 312.524,Z 284.178,A -85,B 0,C 180,E1 -15456.124,E2 -15456.124} C_VEL
LIN {X 0,Y 312.561,Z 284.173,A -85,B 0,C 180,E1 -15460.29,E2 -15460.29} C_VEL
LIN {X 0,Y 312.593,Z 284.173,A -85,B 0,C 180,E1 -15463.007,E2 -15463.007} C_VEL
LIN {X 0,Y 312.68,Z 284.159,A -85,B 0,C 180,E1 -15465.687,E2 -15465.687} C_VEL
LIN {X 0,Y 312.688,Z 284.158,A -85,B 0,C 180,E1 -15469.643,E2 -15469.643} C_VEL
LIN {X 0,Y 312.852,Z 284.137,A -85,B 0,C 180,E1 -15472.255,E2 -15472.255} C_VEL
LIN {X 0,Y 312.702,Z 284.159,A -85,B 0,C 180,E1 -15474.843,E2 -15474.843} C_VEL
LIN {X 0,Y 312.978,Z 284.124,A -85,B 0,C 180,E1 -15478.714,E2 -15478.714} C_VEL
LIN {X 0,Y 312.98,Z 284.124,A -85,B 0,C 180,E1 -15481.288,E2 -15481.288} C_VEL
LIN {X 0,Y 312.704,Z 284.159,A -85,B 0,C 180,E1 -15485.159,E2 -15485.159} C_VEL
LIN {X 0,Y 312.86,Z 284.136,A -85,B 0,C 180,E1 -15487.747,E2 -15487.747} C_VEL
LIN {X 0,Y 312.658,Z 284.161,A -85,B 0,C 180,E1 -15491.673,E2 -15491.673} C_VEL
LIN {X 0,Y 312.689,Z 284.162,A -85,B 0,C 180,E1 -15494.889,E2 -15494.889} C_VEL
LIN {X 0,Y 312.599,Z 284.171,A -85,B 0,C 180,E1 -15499.227,E2 -15499.227} C_VEL
LIN {X 0,Y 312.516,Z 284.183,A -85,B 0,C 180,E1 -15502.782,E2 -15502.782} C_VEL
LIN {X 0,Y 312.588,Z 284.17,A -85,B 0,C 180,E1 -15505.935,E2 -15505.935} C_VEL
LIN {X 0,Y 312.536,Z 284.176,A -85,B 0,C 180,E1 -15509.652,E2 -15509.652} C_VEL
LIN {X 0,Y 312.511,Z 284.179,A -85,B 0,C 180,E1 -15513.691,E2 -15513.691} C_VEL
LIN {X 0,Y 312.512,Z 284.18,A -85,B 0,C 180,E1 -15517.388,E2 -15517.388} C_VEL
LIN {X 0,Y 312.483,Z 284.188,A -85,B 0,C 180,E1 -15520.711,E2 -15520.711} C_VEL
LIN {X 0,Y 312.467,Z 284.186,A -85,B 0,C 180,E1 -15524.208,E2 -15524.208} C_VEL
LIN {X 0,Y 312.48,Z 284.184,A -85,B 0,C 180,E1 -15527.92,E2 -15527.92} C_VEL
LIN {X 0,Y 312.544,Z 284.254,A -85,B 0,C 180,E1 -15529.773,E2 -15529.773} C_VEL
LIN {X 0,Y 316.429,Z 299.907,A -85,B 0,C 180,E1 -15533.621,E2 -15533.621} C_VEL
LIN {X 0,Y 319.086,Z 310.87,A -85,B 0,C 180,E1 -15536.168,E2 -15536.168} C_VEL
LIN {X 0,Y 324.933,Z 327.17,A -85,B 0,C 180,E1 -15537.194,E2 -15537.194} C_VEL
LIN {X 0,Y 329.887,Z 362.182,A -85,B 0,C 180,E1 -15538.749,E2 -15538.749} C_VEL
LIN {X 0,Y 324.272,Z 477.971,A -85,B 0,C 180,E1 -15542.317,E2 -15542.317} C_VEL
LIN {X 0,Y 323.133,Z 493.388,A -85,B 0,C 180,E1 -15543.008,E2 -15543.008} C_VEL
LIN {X 0,Y 321.64,Z 509.175,A -85,B 0,C 180,E1 -15543.973,E2 -15543.973} C_VEL
LIN {X 0,Y 320.088,Z 524.28,A -85,B 0,C 180,E1 -15545.173,E2 -15545.173} C_VEL
LIN {X 0,Y 318.439,Z 538.613,A -85,B 0,C 180,E1 -15546.595,E2 -15546.595} C_VEL
LIN {X 0,Y 316.759,Z 552.011,A -85,B 0,C 180,E1 -15548.22,E2 -15548.22} C_VEL
LIN {X 0,Y 315.168,Z 564.929,A -85,B 0,C 180,E1 -15550.121,E2 -15550.121} C_VEL
LIN {X 0,Y 313.838,Z 575.924,A -85,B 0,C 180,E1 -15552.069,E2 -15552.069} C_VEL
LIN {X 0,Y 312.786,Z 585.218,A -85,B 0,C 180,E1 -15554.025,E2 -15554.025} C_VEL
LIN {X 0,Y 311.937,Z 594.321,A -85,B 0,C 180,E1 -15556.318,E2 -15556.318} C_VEL
LIN {X 0,Y 311.45,Z 600.852,A -85,B 0,C 180,E1 -15558.284,E2 -15558.284} C_VEL
LIN {X 0,Y 311.068,Z 607.887,A -85,B 0,C 180,E1 -15560.902,E2 -15560.902} C_VEL
LIN {X 0,Y 311.015,Z 613.278,A -85,B 0,C 180,E1 -15563.514,E2 -15563.514} C_VEL
LIN {X 0,Y 311.023,Z 615.395,A -85,B 0,C 180,E1 -15564.816,E2 -15564.816} C_VEL
LIN {X 0,Y 310.97,Z 618.518,A -85,B 0,C 180,E1 -15567.411,E2 -15567.411} C_VEL
LIN {X 0,Y 311.117,Z 619.57,A -85,B 0,C 180,E1 -15568.707,E2 -15568.707} C_VEL
LIN {X 0,Y 311.1,Z 620.268,A -85,B 0,C 180,E1 -15570.002,E2 -15570.002} C_VEL
LIN {X 0,Y 311.034,Z 620.623,A -85,B 0,C 180,E1 -15571.296,E2 -15571.296} C_VEL
LIN {X 0,Y 310.836,Z 620.308,A -85,B 0,C 180,E1 -15573.891,E2 -15573.891} C_VEL
LIN {X 0,Y 310.802,Z 618.701,A -85,B 0,C 180,E1 -15576.494,E2 -15576.494} C_VEL
LIN {X 0,Y 310.961,Z 615.824,A -85,B 0,C 180,E1 -15579.104,E2 -15579.104} C_VEL
LIN {X 0,Y 311.495,Z 611.665,A -85,B 0,C 180,E1 -15581.718,E2 -15581.718} C_VEL
LIN {X 0,Y 312.466,Z 606.153,A -85,B 0,C 180,E1 -15584.326,E2 -15584.326} C_VEL
LIN {X 0,Y 314.014,Z 599.186,A -85,B 0,C 180,E1 -15586.917,E2 -15586.917} C_VEL
LIN {X 0,Y 316.139,Z 590.63,A -85,B 0,C 180,E1 -15589.481,E2 -15589.481} C_VEL
LIN {X 0,Y 318.82,Z 580.284,A -85,B 0,C 180,E1 -15592.01,E2 -15592.01} C_VEL
LIN {X 0,Y 321.818,Z 569.504,A -85,B 0,C 180,E1 -15594.173,E2 -15594.173} C_VEL
LIN {X 0,Y 325.32,Z 556.789,A -85,B 0,C 180,E1 -15596.289,E2 -15596.289} C_VEL
LIN {X 0,Y 328.845,Z 543.956,A -85,B 0,C 180,E1 -15598.047,E2 -15598.047} C_VEL
LIN {X 0,Y 332.591,Z 529.717,A -85,B 0,C 180,E1 -15599.661,E2 -15599.661} C_VEL
LIN {X 0,Y 336.292,Z 514.98,A -85,B 0,C 180,E1 -15601.011,E2 -15601.011} C_VEL
LIN {X 0,Y 339.467,Z 501.141,A -85,B 0,C 180,E1 -15602.042,E2 -15602.042} C_VEL
LIN {X 0,Y 343.083,Z 483.708,A -85,B 0,C 180,E1 -15603.054,E2 -15603.054} C_VEL
LIN {X 0,Y 346.125,Z 464.769,A -85,B 0,C 180,E1 -15603.902,E2 -15603.902} C_VEL
LIN {X 0,Y 356.3,Z 393.996,A -85,B 0,C 180,E1 -15606.531,E2 -15606.531} C_VEL
LIN {X 0,Y 360.124,Z 369.796,A -85,B 0,C 180,E1 -15607.454,E2 -15607.454} C_VEL
LIN {X 0,Y 360.552,Z 359.998,A -85,B 0,C 180,E1 -15608.268,E2 -15608.268} C_VEL
LIN {X 0,Y 359.079,Z 354.401,A -85,B 0,C 180,E1 -15609.541,E2 -15609.541} C_VEL
LIN {X 0,Y 357.476,Z 349.107,A -85,B 0,C 180,E1 -15611.221,E2 -15611.221} C_VEL
LIN {X 0,Y 356.188,Z 344.513,A -85,B 0,C 180,E1 -15613.457,E2 -15613.457} C_VEL
LIN {X 0,Y 355.938,Z 342.76,A -85,B 0,C 180,E1 -15614.895,E2 -15614.895} C_VEL
LIN {X 0,Y 356.174,Z 342.404,A -85,B 0,C 180,E1 -15616.895,E2 -15616.895} C_VEL
LIN {X 0,Y 357.773,Z 343.713,A -85,B 0,C 180,E1 -15619.302,E2 -15619.302} C_VEL
LIN {X 0,Y 359.82,Z 346.92,A -85,B 0,C 180,E1 -15621.166,E2 -15621.166} C_VEL
LIN {X 0,Y 361.607,Z 350.193,A -85,B 0,C 180,E1 -15622.416,E2 -15622.416} C_VEL
LIN {X 0,Y 362.368,Z 351.667,A -85,B 0,C 180,E1 -15622.889,E2 -15622.889} C_VEL
LIN {X 0,Y 351.628,Z 417.819,A -85,B 0,C 180,E1 -15625.373,E2 -15625.373} C_VEL
LIN {X 0,Y 346.689,Z 452.757,A -85,B 0,C 180,E1 -15626.746,E2 -15626.746} C_VEL
LIN {X 0,Y 344.137,Z 468.283,A -85,B 0,C 180,E1 -15627.582,E2 -15627.582} C_VEL
LIN {X 0,Y 341.165,Z 483.653,A -85,B 0,C 180,E1 -15628.657,E2 -15628.657} C_VEL
LIN {X 0,Y 338.084,Z 497.776,A -85,B 0,C 180,E1 -15629.9,E2 -15629.9} C_VEL
LIN {X 0,Y 334.59,Z 512.154,A -85,B 0,C 180,E1 -15631.454,E2 -15631.454} C_VEL
LIN {X 0,Y 331.096,Z 525.204,A -85,B 0,C 180,E1 -15633.175,E2 -15633.175} C_VEL
LIN {X 0,Y 327.77,Z 536.412,A -85,B 0,C 180,E1 -15634.945,E2 -15634.945} C_VEL
LIN {X 0,Y 324.456,Z 547.333,A -85,B 0,C 180,E1 -15637.051,E2 -15637.051} C_VEL
LIN {X 0,Y 321.605,Z 556.504,A -85,B 0,C 180,E1 -15639.199,E2 -15639.199} C_VEL
LIN {X 0,Y 318.829,Z 564.872,A -85,B 0,C 180,E1 -15641.58,E2 -15641.58} C_VEL
LIN {X 0,Y 316.596,Z 571.456,A -85,B 0,C 180,E1 -15643.889,E2 -15643.889} C_VEL
LIN {X 0,Y 314.679,Z 577.174,A -85,B 0,C 180,E1 -15646.437,E2 -15646.437} C_VEL
LIN {X 0,Y 313.712,Z 580.485,A -85,B 0,C 180,E1 -15648.367,E2 -15648.367} C_VEL
LIN {X 0,Y 312.609,Z 583.833,A -85,B 0,C 180,E1 -15650.945,E2 -15650.945} C_VEL
LIN {X 0,Y 311.694,Z 585.954,A -85,B 0,C 180,E1 -15653.526,E2 -15653.526} C_VEL
LIN {X 0,Y 311.35,Z 586.837,A -85,B 0,C 180,E1 -15656.116,E2 -15656.116} C_VEL
LIN {X 0,Y 311.084,Z 586.489,A -85,B 0,C 180,E1 -15658.704,E2 -15658.704} C_VEL
LIN {X 0,Y 310.939,Z 584.877,A -85,B 0,C 180,E1 -15661.294,E2 -15661.294} C_VEL
LIN {X 0,Y 311.018,Z 581.99,A -85,B 0,C 180,E1 -15663.886,E2 -15663.886} C_VEL
LIN {X 0,Y 311.191,Z 577.76,A -85,B 0,C 180,E1 -15666.483,E2 -15666.483} C_VEL
LIN {X 0,Y 311.522,Z 572.086,A -85,B 0,C 180,E1 -15669.085,E2 -15669.085} C_VEL
LIN {X 0,Y 312.099,Z 564.812,A -85,B 0,C 180,E1 -15671.692,E2 -15671.692} C_VEL
LIN {X 0,Y 312.995,Z 556.932,A -85,B 0,C 180,E1 -15673.967,E2 -15673.967} C_VEL
LIN {X 0,Y 314.024,Z 547.419,A -85,B 0,C 180,E1 -15676.244,E2 -15676.244} C_VEL
LIN {X 0,Y 315.216,Z 537.708,A -85,B 0,C 180,E1 -15678.187,E2 -15678.187} C_VEL
LIN {X 0,Y 316.628,Z 526.237,A -85,B 0,C 180,E1 -15680.122,E2 -15680.122} C_VEL
LIN {X 0,Y 318.058,Z 513.927,A -85,B 0,C 180,E1 -15681.863,E2 -15681.863} C_VEL
LIN {X 0,Y 319.695,Z 500.131,A -85,B 0,C 180,E1 -15683.48,E2 -15683.48} C_VEL
LIN {X 0,Y 321.208,Z 485.215,A -85,B 0,C 180,E1 -15684.908,E2 -15684.908} C_VEL
LIN {X 0,Y 322.605,Z 469.602,A -85,B 0,C 180,E1 -15686.089,E2 -15686.089} C_VEL
LIN {X 0,Y 323.721,Z 453.536,A -85,B 0,C 180,E1 -15687.025,E2 -15687.025} C_VEL
LIN {X 0,Y 324.649,Z 437.633,A -85,B 0,C 180,E1 -15687.692,E2 -15687.692} C_VEL
LIN {X 0,Y 330.151,Z 324.858,A -85,B 0,C 180,E1 -15691.114,E2 -15691.114} C_VEL
LIN {X 0,Y 314.421,Z 289.131,A -85,B 0,C 180,E1 -15693.563,E2 -15693.563} C_VEL
LIN {X 0,Y 312.527,Z 284.183,A -85,B 0,C 180,E1 -15693.911,E2 -15693.911} C_VEL
LIN {X 0,Y 312.516,Z 284.181,A -85,B 0,C 180,E1 -15697.385,E2 -15697.385} C_VEL
LIN {X 0,Y 312.488,Z 284.183,A -85,B 0,C 180,E1 -15700.708,E2 -15700.708} C_VEL
LIN {X 0,Y 312.451,Z 284.189,A -85,B 0,C 180,E1 -15704.208,E2 -15704.208} C_VEL
